// TIA Portal V17 export
// export: Created 2023-08-28T22:41:32.6164324Z, ExportSetting WithDefaults, DisplayName Totally Integrated Automation Portal, DisplayVersion V17 Update 5, DisplayName TIA Portal Openness, DisplayVersion V17 Update 5, DisplayName TIA Portal Teamcenter Gateway, DisplayVersion V17 Update 5, DisplayName TIA Portal Version Control Interface, DisplayVersion V17, DisplayName Simotion SCOUT TIA, DisplayVersion 5.4.3.0, DisplayName TIA Portal Test Suite Advanced, DisplayVersion V17 Update 1, DisplayName SIMOCODE ES, DisplayVersion V17 Update 5, DisplayName SINAMICS Startdrive Advanced, DisplayVersion V17 SP1, DisplayName SINAMICS Startdrive G130, G150, S120, S150, SINAMICS MV, S210, DisplayVersion V17 SP1, DisplayName SINAMICS Startdrive G110M, G120, G120C, G120D, G120P, G115D, DisplayVersion V17 SP1, DisplayName SIRIUS Safety ES, DisplayVersion V17 Update 5, DisplayName STEP 7 Professional, DisplayVersion V17 Update 5, DisplayName STEP 7 CFC, DisplayVersion V17 Update 1, DisplayName STEP 7 Safety, DisplayVersion V17, DisplayName WinCC Advanced, DisplayVersion V17 Update 5, DisplayName SIMATIC Visualization Architect, DisplayVersion V17 Update 5
DATA_BLOCK "n0005-zp001-el001-k40001_SN50_1"   // DB1001, F_DB
VERSION : 0.1
// stored: AutoNumber true, DBAccessibleFromOPCUA true, DBAccessibleFromWebserver true, InstanceOfName 00_Push-Button_Input, InstanceOfType FB
"00_Push-Button_Input"
   // VAR_INPUT
   //    IN_1 : Bool;
   //    IN_2 : Bool;
   //    IN_3 : Bool;
   //    IN_4 : Bool;
   //    ON_Tristate : Bool;
   //    ON_Lamp : Bool;
   //    Reset : Bool;
   //    REAC_DELAY { ExternalWritable := 'False'} : Time;
   //    Bypass_ET200 : Bool;
   // END_VAR
   // VAR_OUTPUT
   //    OUT_1 : Bool;
   //    OUT_2 : Bool;
   //    OUT_3 : Bool;
   //    OUT_4 : Bool;
   //    Diag_1 : Bool;
   //    Diag_2 : Bool;
   //    Diag_3 : Bool;
   //    Diag_4 : Bool;
   //    Lamp_1 : Bool;
   //    Lamp_2 : Bool;
   //    Lamp_3 : Bool;
   //    Lamp_4 : Bool;
   // END_VAR
   // VAR
   //    ESTOP_1 { S7_SetPoint := 'True'} : ESTOP1;
   //    ESTOP_2 { S7_SetPoint := 'True'} : ESTOP1;
   //    ESTOP_3 { S7_SetPoint := 'True'} : ESTOP1;
   //    ESTOP_4 { S7_SetPoint := 'True'} : ESTOP1;
   //    TON_1 { ExternalWritable := 'False'} : TON;
   //    TON_2 { ExternalWritable := 'False'} : TON;
   //    TON_3 { ExternalWritable := 'False'} : TON;
   //    TON_4 { ExternalWritable := 'False'} : TON;
   // END_VAR
BEGIN
END_DATA_BLOCK

DATA_BLOCK "n0013-uf317-xn10_SN50_1"   // DB1002, F_DB
VERSION : 0.1
// stored: AutoNumber true, DBAccessibleFromOPCUA true, DBAccessibleFromWebserver true, InstanceOfName 00_Push-Button_Input, InstanceOfType FB
"00_Push-Button_Input"
   // VAR_INPUT
   //    IN_1 : Bool;
   //    IN_2 : Bool;
   //    IN_3 : Bool;
   //    IN_4 : Bool;
   //    ON_Tristate : Bool;
   //    ON_Lamp : Bool;
   //    Reset : Bool;
   //    REAC_DELAY { ExternalWritable := 'False'} : Time;
   //    Bypass_ET200 : Bool;
   // END_VAR
   // VAR_OUTPUT
   //    OUT_1 : Bool;
   //    OUT_2 : Bool;
   //    OUT_3 : Bool;
   //    OUT_4 : Bool;
   //    Diag_1 : Bool;
   //    Diag_2 : Bool;
   //    Diag_3 : Bool;
   //    Diag_4 : Bool;
   //    Lamp_1 : Bool;
   //    Lamp_2 : Bool;
   //    Lamp_3 : Bool;
   //    Lamp_4 : Bool;
   // END_VAR
   // VAR
   //    ESTOP_1 { S7_SetPoint := 'True'} : ESTOP1;
   //    ESTOP_2 { S7_SetPoint := 'True'} : ESTOP1;
   //    ESTOP_3 { S7_SetPoint := 'True'} : ESTOP1;
   //    ESTOP_4 { S7_SetPoint := 'True'} : ESTOP1;
   //    TON_1 { ExternalWritable := 'False'} : TON;
   //    TON_2 { ExternalWritable := 'False'} : TON;
   //    TON_3 { ExternalWritable := 'False'} : TON;
   //    TON_4 { ExternalWritable := 'False'} : TON;
   // END_VAR
BEGIN
END_DATA_BLOCK

DATA_BLOCK "n0013-uf317-xn10_SN50_2"   // DB1003, F_DB
VERSION : 0.1
// stored: AutoNumber true, DBAccessibleFromOPCUA true, DBAccessibleFromWebserver true, InstanceOfName 00_Push-Button_Input, InstanceOfType FB
"00_Push-Button_Input"
   // VAR_INPUT
   //    IN_1 : Bool;
   //    IN_2 : Bool;
   //    IN_3 : Bool;
   //    IN_4 : Bool;
   //    ON_Tristate : Bool;
   //    ON_Lamp : Bool;
   //    Reset : Bool;
   //    REAC_DELAY { ExternalWritable := 'False'} : Time;
   //    Bypass_ET200 : Bool;
   // END_VAR
   // VAR_OUTPUT
   //    OUT_1 : Bool;
   //    OUT_2 : Bool;
   //    OUT_3 : Bool;
   //    OUT_4 : Bool;
   //    Diag_1 : Bool;
   //    Diag_2 : Bool;
   //    Diag_3 : Bool;
   //    Diag_4 : Bool;
   //    Lamp_1 : Bool;
   //    Lamp_2 : Bool;
   //    Lamp_3 : Bool;
   //    Lamp_4 : Bool;
   // END_VAR
   // VAR
   //    ESTOP_1 { S7_SetPoint := 'True'} : ESTOP1;
   //    ESTOP_2 { S7_SetPoint := 'True'} : ESTOP1;
   //    ESTOP_3 { S7_SetPoint := 'True'} : ESTOP1;
   //    ESTOP_4 { S7_SetPoint := 'True'} : ESTOP1;
   //    TON_1 { ExternalWritable := 'False'} : TON;
   //    TON_2 { ExternalWritable := 'False'} : TON;
   //    TON_3 { ExternalWritable := 'False'} : TON;
   //    TON_4 { ExternalWritable := 'False'} : TON;
   // END_VAR
BEGIN
END_DATA_BLOCK

DATA_BLOCK "n0015-uc16-el001-k30001_SN50_1"   // DB1004, F_DB
VERSION : 0.1
// stored: AutoNumber true, DBAccessibleFromOPCUA true, DBAccessibleFromWebserver true, InstanceOfName 00_Push-Button_Input, InstanceOfType FB
"00_Push-Button_Input"
   // VAR_INPUT
   //    IN_1 : Bool;
   //    IN_2 : Bool;
   //    IN_3 : Bool;
   //    IN_4 : Bool;
   //    ON_Tristate : Bool;
   //    ON_Lamp : Bool;
   //    Reset : Bool;
   //    REAC_DELAY { ExternalWritable := 'False'} : Time;
   //    Bypass_ET200 : Bool;
   // END_VAR
   // VAR_OUTPUT
   //    OUT_1 : Bool;
   //    OUT_2 : Bool;
   //    OUT_3 : Bool;
   //    OUT_4 : Bool;
   //    Diag_1 : Bool;
   //    Diag_2 : Bool;
   //    Diag_3 : Bool;
   //    Diag_4 : Bool;
   //    Lamp_1 : Bool;
   //    Lamp_2 : Bool;
   //    Lamp_3 : Bool;
   //    Lamp_4 : Bool;
   // END_VAR
   // VAR
   //    ESTOP_1 { S7_SetPoint := 'True'} : ESTOP1;
   //    ESTOP_2 { S7_SetPoint := 'True'} : ESTOP1;
   //    ESTOP_3 { S7_SetPoint := 'True'} : ESTOP1;
   //    ESTOP_4 { S7_SetPoint := 'True'} : ESTOP1;
   //    TON_1 { ExternalWritable := 'False'} : TON;
   //    TON_2 { ExternalWritable := 'False'} : TON;
   //    TON_3 { ExternalWritable := 'False'} : TON;
   //    TON_4 { ExternalWritable := 'False'} : TON;
   // END_VAR
BEGIN
END_DATA_BLOCK

DATA_BLOCK "n0015-uc16-el001-k30001_SN50_2"   // DB1005, F_DB
VERSION : 0.1
// stored: AutoNumber true, DBAccessibleFromOPCUA true, DBAccessibleFromWebserver true, InstanceOfName 00_Push-Button_Input, InstanceOfType FB
"00_Push-Button_Input"
   // VAR_INPUT
   //    IN_1 : Bool;
   //    IN_2 : Bool;
   //    IN_3 : Bool;
   //    IN_4 : Bool;
   //    ON_Tristate : Bool;
   //    ON_Lamp : Bool;
   //    Reset : Bool;
   //    REAC_DELAY { ExternalWritable := 'False'} : Time;
   //    Bypass_ET200 : Bool;
   // END_VAR
   // VAR_OUTPUT
   //    OUT_1 : Bool;
   //    OUT_2 : Bool;
   //    OUT_3 : Bool;
   //    OUT_4 : Bool;
   //    Diag_1 : Bool;
   //    Diag_2 : Bool;
   //    Diag_3 : Bool;
   //    Diag_4 : Bool;
   //    Lamp_1 : Bool;
   //    Lamp_2 : Bool;
   //    Lamp_3 : Bool;
   //    Lamp_4 : Bool;
   // END_VAR
   // VAR
   //    ESTOP_1 { S7_SetPoint := 'True'} : ESTOP1;
   //    ESTOP_2 { S7_SetPoint := 'True'} : ESTOP1;
   //    ESTOP_3 { S7_SetPoint := 'True'} : ESTOP1;
   //    ESTOP_4 { S7_SetPoint := 'True'} : ESTOP1;
   //    TON_1 { ExternalWritable := 'False'} : TON;
   //    TON_2 { ExternalWritable := 'False'} : TON;
   //    TON_3 { ExternalWritable := 'False'} : TON;
   //    TON_4 { ExternalWritable := 'False'} : TON;
   // END_VAR
BEGIN
END_DATA_BLOCK

DATA_BLOCK "n0015-uc16-el001-k30001_SN50_3"   // DB1006, F_DB
VERSION : 0.1
// stored: AutoNumber true, DBAccessibleFromOPCUA true, DBAccessibleFromWebserver true, InstanceOfName 00_Push-Button_Input, InstanceOfType FB
"00_Push-Button_Input"
   // VAR_INPUT
   //    IN_1 : Bool;
   //    IN_2 : Bool;
   //    IN_3 : Bool;
   //    IN_4 : Bool;
   //    ON_Tristate : Bool;
   //    ON_Lamp : Bool;
   //    Reset : Bool;
   //    REAC_DELAY { ExternalWritable := 'False'} : Time;
   //    Bypass_ET200 : Bool;
   // END_VAR
   // VAR_OUTPUT
   //    OUT_1 : Bool;
   //    OUT_2 : Bool;
   //    OUT_3 : Bool;
   //    OUT_4 : Bool;
   //    Diag_1 : Bool;
   //    Diag_2 : Bool;
   //    Diag_3 : Bool;
   //    Diag_4 : Bool;
   //    Lamp_1 : Bool;
   //    Lamp_2 : Bool;
   //    Lamp_3 : Bool;
   //    Lamp_4 : Bool;
   // END_VAR
   // VAR
   //    ESTOP_1 { S7_SetPoint := 'True'} : ESTOP1;
   //    ESTOP_2 { S7_SetPoint := 'True'} : ESTOP1;
   //    ESTOP_3 { S7_SetPoint := 'True'} : ESTOP1;
   //    ESTOP_4 { S7_SetPoint := 'True'} : ESTOP1;
   //    TON_1 { ExternalWritable := 'False'} : TON;
   //    TON_2 { ExternalWritable := 'False'} : TON;
   //    TON_3 { ExternalWritable := 'False'} : TON;
   //    TON_4 { ExternalWritable := 'False'} : TON;
   // END_VAR
BEGIN
END_DATA_BLOCK

DATA_BLOCK "n0016-uc164-xn10_SN50_1"   // DB1007, F_DB
VERSION : 0.1
// stored: AutoNumber true, DBAccessibleFromOPCUA true, DBAccessibleFromWebserver true, InstanceOfName 00_Push-Button_Input, InstanceOfType FB
"00_Push-Button_Input"
   // VAR_INPUT
   //    IN_1 : Bool;
   //    IN_2 : Bool;
   //    IN_3 : Bool;
   //    IN_4 : Bool;
   //    ON_Tristate : Bool;
   //    ON_Lamp : Bool;
   //    Reset : Bool;
   //    REAC_DELAY { ExternalWritable := 'False'} : Time;
   //    Bypass_ET200 : Bool;
   // END_VAR
   // VAR_OUTPUT
   //    OUT_1 : Bool;
   //    OUT_2 : Bool;
   //    OUT_3 : Bool;
   //    OUT_4 : Bool;
   //    Diag_1 : Bool;
   //    Diag_2 : Bool;
   //    Diag_3 : Bool;
   //    Diag_4 : Bool;
   //    Lamp_1 : Bool;
   //    Lamp_2 : Bool;
   //    Lamp_3 : Bool;
   //    Lamp_4 : Bool;
   // END_VAR
   // VAR
   //    ESTOP_1 { S7_SetPoint := 'True'} : ESTOP1;
   //    ESTOP_2 { S7_SetPoint := 'True'} : ESTOP1;
   //    ESTOP_3 { S7_SetPoint := 'True'} : ESTOP1;
   //    ESTOP_4 { S7_SetPoint := 'True'} : ESTOP1;
   //    TON_1 { ExternalWritable := 'False'} : TON;
   //    TON_2 { ExternalWritable := 'False'} : TON;
   //    TON_3 { ExternalWritable := 'False'} : TON;
   //    TON_4 { ExternalWritable := 'False'} : TON;
   // END_VAR
BEGIN
END_DATA_BLOCK

DATA_BLOCK "n0016-uc164-xn10_SN50_2"   // DB1008, F_DB
VERSION : 0.1
// stored: AutoNumber true, DBAccessibleFromOPCUA true, DBAccessibleFromWebserver true, InstanceOfName 00_Push-Button_Input, InstanceOfType FB
"00_Push-Button_Input"
   // VAR_INPUT
   //    IN_1 : Bool;
   //    IN_2 : Bool;
   //    IN_3 : Bool;
   //    IN_4 : Bool;
   //    ON_Tristate : Bool;
   //    ON_Lamp : Bool;
   //    Reset : Bool;
   //    REAC_DELAY { ExternalWritable := 'False'} : Time;
   //    Bypass_ET200 : Bool;
   // END_VAR
   // VAR_OUTPUT
   //    OUT_1 : Bool;
   //    OUT_2 : Bool;
   //    OUT_3 : Bool;
   //    OUT_4 : Bool;
   //    Diag_1 : Bool;
   //    Diag_2 : Bool;
   //    Diag_3 : Bool;
   //    Diag_4 : Bool;
   //    Lamp_1 : Bool;
   //    Lamp_2 : Bool;
   //    Lamp_3 : Bool;
   //    Lamp_4 : Bool;
   // END_VAR
   // VAR
   //    ESTOP_1 { S7_SetPoint := 'True'} : ESTOP1;
   //    ESTOP_2 { S7_SetPoint := 'True'} : ESTOP1;
   //    ESTOP_3 { S7_SetPoint := 'True'} : ESTOP1;
   //    ESTOP_4 { S7_SetPoint := 'True'} : ESTOP1;
   //    TON_1 { ExternalWritable := 'False'} : TON;
   //    TON_2 { ExternalWritable := 'False'} : TON;
   //    TON_3 { ExternalWritable := 'False'} : TON;
   //    TON_4 { ExternalWritable := 'False'} : TON;
   // END_VAR
BEGIN
END_DATA_BLOCK

DATA_BLOCK "n0020-uc15-el001-k30001_SN50_1"   // DB1009, F_DB
VERSION : 0.1
// stored: AutoNumber true, DBAccessibleFromOPCUA true, DBAccessibleFromWebserver true, InstanceOfName 00_Push-Button_Input, InstanceOfType FB
"00_Push-Button_Input"
   // VAR_INPUT
   //    IN_1 : Bool;
   //    IN_2 : Bool;
   //    IN_3 : Bool;
   //    IN_4 : Bool;
   //    ON_Tristate : Bool;
   //    ON_Lamp : Bool;
   //    Reset : Bool;
   //    REAC_DELAY { ExternalWritable := 'False'} : Time;
   //    Bypass_ET200 : Bool;
   // END_VAR
   // VAR_OUTPUT
   //    OUT_1 : Bool;
   //    OUT_2 : Bool;
   //    OUT_3 : Bool;
   //    OUT_4 : Bool;
   //    Diag_1 : Bool;
   //    Diag_2 : Bool;
   //    Diag_3 : Bool;
   //    Diag_4 : Bool;
   //    Lamp_1 : Bool;
   //    Lamp_2 : Bool;
   //    Lamp_3 : Bool;
   //    Lamp_4 : Bool;
   // END_VAR
   // VAR
   //    ESTOP_1 { S7_SetPoint := 'True'} : ESTOP1;
   //    ESTOP_2 { S7_SetPoint := 'True'} : ESTOP1;
   //    ESTOP_3 { S7_SetPoint := 'True'} : ESTOP1;
   //    ESTOP_4 { S7_SetPoint := 'True'} : ESTOP1;
   //    TON_1 { ExternalWritable := 'False'} : TON;
   //    TON_2 { ExternalWritable := 'False'} : TON;
   //    TON_3 { ExternalWritable := 'False'} : TON;
   //    TON_4 { ExternalWritable := 'False'} : TON;
   // END_VAR
BEGIN
END_DATA_BLOCK

DATA_BLOCK "n0020-uc15-el001-k30001_SN50_2"   // DB1010, F_DB
VERSION : 0.1
// stored: AutoNumber true, DBAccessibleFromOPCUA true, DBAccessibleFromWebserver true, InstanceOfName 00_Push-Button_Input, InstanceOfType FB
"00_Push-Button_Input"
   // VAR_INPUT
   //    IN_1 : Bool;
   //    IN_2 : Bool;
   //    IN_3 : Bool;
   //    IN_4 : Bool;
   //    ON_Tristate : Bool;
   //    ON_Lamp : Bool;
   //    Reset : Bool;
   //    REAC_DELAY { ExternalWritable := 'False'} : Time;
   //    Bypass_ET200 : Bool;
   // END_VAR
   // VAR_OUTPUT
   //    OUT_1 : Bool;
   //    OUT_2 : Bool;
   //    OUT_3 : Bool;
   //    OUT_4 : Bool;
   //    Diag_1 : Bool;
   //    Diag_2 : Bool;
   //    Diag_3 : Bool;
   //    Diag_4 : Bool;
   //    Lamp_1 : Bool;
   //    Lamp_2 : Bool;
   //    Lamp_3 : Bool;
   //    Lamp_4 : Bool;
   // END_VAR
   // VAR
   //    ESTOP_1 { S7_SetPoint := 'True'} : ESTOP1;
   //    ESTOP_2 { S7_SetPoint := 'True'} : ESTOP1;
   //    ESTOP_3 { S7_SetPoint := 'True'} : ESTOP1;
   //    ESTOP_4 { S7_SetPoint := 'True'} : ESTOP1;
   //    TON_1 { ExternalWritable := 'False'} : TON;
   //    TON_2 { ExternalWritable := 'False'} : TON;
   //    TON_3 { ExternalWritable := 'False'} : TON;
   //    TON_4 { ExternalWritable := 'False'} : TON;
   // END_VAR
BEGIN
END_DATA_BLOCK

DATA_BLOCK "n0020-uc15-el001-k30001_SN50_3"   // DB1011, F_DB
VERSION : 0.1
// stored: AutoNumber true, DBAccessibleFromOPCUA true, DBAccessibleFromWebserver true, InstanceOfName 00_Push-Button_Input, InstanceOfType FB
"00_Push-Button_Input"
   // VAR_INPUT
   //    IN_1 : Bool;
   //    IN_2 : Bool;
   //    IN_3 : Bool;
   //    IN_4 : Bool;
   //    ON_Tristate : Bool;
   //    ON_Lamp : Bool;
   //    Reset : Bool;
   //    REAC_DELAY { ExternalWritable := 'False'} : Time;
   //    Bypass_ET200 : Bool;
   // END_VAR
   // VAR_OUTPUT
   //    OUT_1 : Bool;
   //    OUT_2 : Bool;
   //    OUT_3 : Bool;
   //    OUT_4 : Bool;
   //    Diag_1 : Bool;
   //    Diag_2 : Bool;
   //    Diag_3 : Bool;
   //    Diag_4 : Bool;
   //    Lamp_1 : Bool;
   //    Lamp_2 : Bool;
   //    Lamp_3 : Bool;
   //    Lamp_4 : Bool;
   // END_VAR
   // VAR
   //    ESTOP_1 { S7_SetPoint := 'True'} : ESTOP1;
   //    ESTOP_2 { S7_SetPoint := 'True'} : ESTOP1;
   //    ESTOP_3 { S7_SetPoint := 'True'} : ESTOP1;
   //    ESTOP_4 { S7_SetPoint := 'True'} : ESTOP1;
   //    TON_1 { ExternalWritable := 'False'} : TON;
   //    TON_2 { ExternalWritable := 'False'} : TON;
   //    TON_3 { ExternalWritable := 'False'} : TON;
   //    TON_4 { ExternalWritable := 'False'} : TON;
   // END_VAR
BEGIN
END_DATA_BLOCK

DATA_BLOCK "n0023-uc154-xn10_SN50_1"   // DB1012, F_DB
VERSION : 0.1
// stored: AutoNumber true, DBAccessibleFromOPCUA true, DBAccessibleFromWebserver true, InstanceOfName 00_Push-Button_Input, InstanceOfType FB
"00_Push-Button_Input"
   // VAR_INPUT
   //    IN_1 : Bool;
   //    IN_2 : Bool;
   //    IN_3 : Bool;
   //    IN_4 : Bool;
   //    ON_Tristate : Bool;
   //    ON_Lamp : Bool;
   //    Reset : Bool;
   //    REAC_DELAY { ExternalWritable := 'False'} : Time;
   //    Bypass_ET200 : Bool;
   // END_VAR
   // VAR_OUTPUT
   //    OUT_1 : Bool;
   //    OUT_2 : Bool;
   //    OUT_3 : Bool;
   //    OUT_4 : Bool;
   //    Diag_1 : Bool;
   //    Diag_2 : Bool;
   //    Diag_3 : Bool;
   //    Diag_4 : Bool;
   //    Lamp_1 : Bool;
   //    Lamp_2 : Bool;
   //    Lamp_3 : Bool;
   //    Lamp_4 : Bool;
   // END_VAR
   // VAR
   //    ESTOP_1 { S7_SetPoint := 'True'} : ESTOP1;
   //    ESTOP_2 { S7_SetPoint := 'True'} : ESTOP1;
   //    ESTOP_3 { S7_SetPoint := 'True'} : ESTOP1;
   //    ESTOP_4 { S7_SetPoint := 'True'} : ESTOP1;
   //    TON_1 { ExternalWritable := 'False'} : TON;
   //    TON_2 { ExternalWritable := 'False'} : TON;
   //    TON_3 { ExternalWritable := 'False'} : TON;
   //    TON_4 { ExternalWritable := 'False'} : TON;
   // END_VAR
BEGIN
END_DATA_BLOCK

DATA_BLOCK "n0023-uc154-xn10_SN50_2"   // DB1013, F_DB
VERSION : 0.1
// stored: AutoNumber true, DBAccessibleFromOPCUA true, DBAccessibleFromWebserver true, InstanceOfName 00_Push-Button_Input, InstanceOfType FB
"00_Push-Button_Input"
   // VAR_INPUT
   //    IN_1 : Bool;
   //    IN_2 : Bool;
   //    IN_3 : Bool;
   //    IN_4 : Bool;
   //    ON_Tristate : Bool;
   //    ON_Lamp : Bool;
   //    Reset : Bool;
   //    REAC_DELAY { ExternalWritable := 'False'} : Time;
   //    Bypass_ET200 : Bool;
   // END_VAR
   // VAR_OUTPUT
   //    OUT_1 : Bool;
   //    OUT_2 : Bool;
   //    OUT_3 : Bool;
   //    OUT_4 : Bool;
   //    Diag_1 : Bool;
   //    Diag_2 : Bool;
   //    Diag_3 : Bool;
   //    Diag_4 : Bool;
   //    Lamp_1 : Bool;
   //    Lamp_2 : Bool;
   //    Lamp_3 : Bool;
   //    Lamp_4 : Bool;
   // END_VAR
   // VAR
   //    ESTOP_1 { S7_SetPoint := 'True'} : ESTOP1;
   //    ESTOP_2 { S7_SetPoint := 'True'} : ESTOP1;
   //    ESTOP_3 { S7_SetPoint := 'True'} : ESTOP1;
   //    ESTOP_4 { S7_SetPoint := 'True'} : ESTOP1;
   //    TON_1 { ExternalWritable := 'False'} : TON;
   //    TON_2 { ExternalWritable := 'False'} : TON;
   //    TON_3 { ExternalWritable := 'False'} : TON;
   //    TON_4 { ExternalWritable := 'False'} : TON;
   // END_VAR
BEGIN
END_DATA_BLOCK

DATA_BLOCK "n0021-icg11-el001-k30001_SN50_1"   // DB1014, F_DB
VERSION : 0.1
// stored: AutoNumber true, DBAccessibleFromOPCUA true, DBAccessibleFromWebserver true, InstanceOfName 00_Push-Button_Input, InstanceOfType FB
"00_Push-Button_Input"
   // VAR_INPUT
   //    IN_1 : Bool;
   //    IN_2 : Bool;
   //    IN_3 : Bool;
   //    IN_4 : Bool;
   //    ON_Tristate : Bool;
   //    ON_Lamp : Bool;
   //    Reset : Bool;
   //    REAC_DELAY { ExternalWritable := 'False'} : Time;
   //    Bypass_ET200 : Bool;
   // END_VAR
   // VAR_OUTPUT
   //    OUT_1 : Bool;
   //    OUT_2 : Bool;
   //    OUT_3 : Bool;
   //    OUT_4 : Bool;
   //    Diag_1 : Bool;
   //    Diag_2 : Bool;
   //    Diag_3 : Bool;
   //    Diag_4 : Bool;
   //    Lamp_1 : Bool;
   //    Lamp_2 : Bool;
   //    Lamp_3 : Bool;
   //    Lamp_4 : Bool;
   // END_VAR
   // VAR
   //    ESTOP_1 { S7_SetPoint := 'True'} : ESTOP1;
   //    ESTOP_2 { S7_SetPoint := 'True'} : ESTOP1;
   //    ESTOP_3 { S7_SetPoint := 'True'} : ESTOP1;
   //    ESTOP_4 { S7_SetPoint := 'True'} : ESTOP1;
   //    TON_1 { ExternalWritable := 'False'} : TON;
   //    TON_2 { ExternalWritable := 'False'} : TON;
   //    TON_3 { ExternalWritable := 'False'} : TON;
   //    TON_4 { ExternalWritable := 'False'} : TON;
   // END_VAR
BEGIN
END_DATA_BLOCK

DATA_BLOCK "n0021-icg11-el001-k30001_SN50_2"   // DB1015, F_DB
VERSION : 0.1
// stored: AutoNumber true, DBAccessibleFromOPCUA true, DBAccessibleFromWebserver true, InstanceOfName 00_Push-Button_Input, InstanceOfType FB
"00_Push-Button_Input"
   // VAR_INPUT
   //    IN_1 : Bool;
   //    IN_2 : Bool;
   //    IN_3 : Bool;
   //    IN_4 : Bool;
   //    ON_Tristate : Bool;
   //    ON_Lamp : Bool;
   //    Reset : Bool;
   //    REAC_DELAY { ExternalWritable := 'False'} : Time;
   //    Bypass_ET200 : Bool;
   // END_VAR
   // VAR_OUTPUT
   //    OUT_1 : Bool;
   //    OUT_2 : Bool;
   //    OUT_3 : Bool;
   //    OUT_4 : Bool;
   //    Diag_1 : Bool;
   //    Diag_2 : Bool;
   //    Diag_3 : Bool;
   //    Diag_4 : Bool;
   //    Lamp_1 : Bool;
   //    Lamp_2 : Bool;
   //    Lamp_3 : Bool;
   //    Lamp_4 : Bool;
   // END_VAR
   // VAR
   //    ESTOP_1 { S7_SetPoint := 'True'} : ESTOP1;
   //    ESTOP_2 { S7_SetPoint := 'True'} : ESTOP1;
   //    ESTOP_3 { S7_SetPoint := 'True'} : ESTOP1;
   //    ESTOP_4 { S7_SetPoint := 'True'} : ESTOP1;
   //    TON_1 { ExternalWritable := 'False'} : TON;
   //    TON_2 { ExternalWritable := 'False'} : TON;
   //    TON_3 { ExternalWritable := 'False'} : TON;
   //    TON_4 { ExternalWritable := 'False'} : TON;
   // END_VAR
BEGIN
END_DATA_BLOCK

DATA_BLOCK "n0021-icg11-el001-k30001_SN50_3"   // DB1016, F_DB
VERSION : 0.1
// stored: AutoNumber true, DBAccessibleFromOPCUA true, DBAccessibleFromWebserver true, InstanceOfName 00_Push-Button_Input, InstanceOfType FB
"00_Push-Button_Input"
   // VAR_INPUT
   //    IN_1 : Bool;
   //    IN_2 : Bool;
   //    IN_3 : Bool;
   //    IN_4 : Bool;
   //    ON_Tristate : Bool;
   //    ON_Lamp : Bool;
   //    Reset : Bool;
   //    REAC_DELAY { ExternalWritable := 'False'} : Time;
   //    Bypass_ET200 : Bool;
   // END_VAR
   // VAR_OUTPUT
   //    OUT_1 : Bool;
   //    OUT_2 : Bool;
   //    OUT_3 : Bool;
   //    OUT_4 : Bool;
   //    Diag_1 : Bool;
   //    Diag_2 : Bool;
   //    Diag_3 : Bool;
   //    Diag_4 : Bool;
   //    Lamp_1 : Bool;
   //    Lamp_2 : Bool;
   //    Lamp_3 : Bool;
   //    Lamp_4 : Bool;
   // END_VAR
   // VAR
   //    ESTOP_1 { S7_SetPoint := 'True'} : ESTOP1;
   //    ESTOP_2 { S7_SetPoint := 'True'} : ESTOP1;
   //    ESTOP_3 { S7_SetPoint := 'True'} : ESTOP1;
   //    ESTOP_4 { S7_SetPoint := 'True'} : ESTOP1;
   //    TON_1 { ExternalWritable := 'False'} : TON;
   //    TON_2 { ExternalWritable := 'False'} : TON;
   //    TON_3 { ExternalWritable := 'False'} : TON;
   //    TON_4 { ExternalWritable := 'False'} : TON;
   // END_VAR
BEGIN
END_DATA_BLOCK

DATA_BLOCK "n0021-icg11-el001-k30001_SN50_4"   // DB1017, F_DB
VERSION : 0.1
// stored: AutoNumber true, DBAccessibleFromOPCUA true, DBAccessibleFromWebserver true, InstanceOfName 00_Push-Button_Input, InstanceOfType FB
"00_Push-Button_Input"
   // VAR_INPUT
   //    IN_1 : Bool;
   //    IN_2 : Bool;
   //    IN_3 : Bool;
   //    IN_4 : Bool;
   //    ON_Tristate : Bool;
   //    ON_Lamp : Bool;
   //    Reset : Bool;
   //    REAC_DELAY { ExternalWritable := 'False'} : Time;
   //    Bypass_ET200 : Bool;
   // END_VAR
   // VAR_OUTPUT
   //    OUT_1 : Bool;
   //    OUT_2 : Bool;
   //    OUT_3 : Bool;
   //    OUT_4 : Bool;
   //    Diag_1 : Bool;
   //    Diag_2 : Bool;
   //    Diag_3 : Bool;
   //    Diag_4 : Bool;
   //    Lamp_1 : Bool;
   //    Lamp_2 : Bool;
   //    Lamp_3 : Bool;
   //    Lamp_4 : Bool;
   // END_VAR
   // VAR
   //    ESTOP_1 { S7_SetPoint := 'True'} : ESTOP1;
   //    ESTOP_2 { S7_SetPoint := 'True'} : ESTOP1;
   //    ESTOP_3 { S7_SetPoint := 'True'} : ESTOP1;
   //    ESTOP_4 { S7_SetPoint := 'True'} : ESTOP1;
   //    TON_1 { ExternalWritable := 'False'} : TON;
   //    TON_2 { ExternalWritable := 'False'} : TON;
   //    TON_3 { ExternalWritable := 'False'} : TON;
   //    TON_4 { ExternalWritable := 'False'} : TON;
   // END_VAR
BEGIN
END_DATA_BLOCK

DATA_BLOCK "n0022-icg21-el001-k30001_SN50_1"   // DB1018, F_DB
VERSION : 0.1
// stored: AutoNumber true, DBAccessibleFromOPCUA true, DBAccessibleFromWebserver true, InstanceOfName 00_Push-Button_Input, InstanceOfType FB
"00_Push-Button_Input"
   // VAR_INPUT
   //    IN_1 : Bool;
   //    IN_2 : Bool;
   //    IN_3 : Bool;
   //    IN_4 : Bool;
   //    ON_Tristate : Bool;
   //    ON_Lamp : Bool;
   //    Reset : Bool;
   //    REAC_DELAY { ExternalWritable := 'False'} : Time;
   //    Bypass_ET200 : Bool;
   // END_VAR
   // VAR_OUTPUT
   //    OUT_1 : Bool;
   //    OUT_2 : Bool;
   //    OUT_3 : Bool;
   //    OUT_4 : Bool;
   //    Diag_1 : Bool;
   //    Diag_2 : Bool;
   //    Diag_3 : Bool;
   //    Diag_4 : Bool;
   //    Lamp_1 : Bool;
   //    Lamp_2 : Bool;
   //    Lamp_3 : Bool;
   //    Lamp_4 : Bool;
   // END_VAR
   // VAR
   //    ESTOP_1 { S7_SetPoint := 'True'} : ESTOP1;
   //    ESTOP_2 { S7_SetPoint := 'True'} : ESTOP1;
   //    ESTOP_3 { S7_SetPoint := 'True'} : ESTOP1;
   //    ESTOP_4 { S7_SetPoint := 'True'} : ESTOP1;
   //    TON_1 { ExternalWritable := 'False'} : TON;
   //    TON_2 { ExternalWritable := 'False'} : TON;
   //    TON_3 { ExternalWritable := 'False'} : TON;
   //    TON_4 { ExternalWritable := 'False'} : TON;
   // END_VAR
BEGIN
END_DATA_BLOCK

DATA_BLOCK "n0022-icg21-el001-k30001_SN50_2"   // DB1019, F_DB
VERSION : 0.1
// stored: AutoNumber true, DBAccessibleFromOPCUA true, DBAccessibleFromWebserver true, InstanceOfName 00_Push-Button_Input, InstanceOfType FB
"00_Push-Button_Input"
   // VAR_INPUT
   //    IN_1 : Bool;
   //    IN_2 : Bool;
   //    IN_3 : Bool;
   //    IN_4 : Bool;
   //    ON_Tristate : Bool;
   //    ON_Lamp : Bool;
   //    Reset : Bool;
   //    REAC_DELAY { ExternalWritable := 'False'} : Time;
   //    Bypass_ET200 : Bool;
   // END_VAR
   // VAR_OUTPUT
   //    OUT_1 : Bool;
   //    OUT_2 : Bool;
   //    OUT_3 : Bool;
   //    OUT_4 : Bool;
   //    Diag_1 : Bool;
   //    Diag_2 : Bool;
   //    Diag_3 : Bool;
   //    Diag_4 : Bool;
   //    Lamp_1 : Bool;
   //    Lamp_2 : Bool;
   //    Lamp_3 : Bool;
   //    Lamp_4 : Bool;
   // END_VAR
   // VAR
   //    ESTOP_1 { S7_SetPoint := 'True'} : ESTOP1;
   //    ESTOP_2 { S7_SetPoint := 'True'} : ESTOP1;
   //    ESTOP_3 { S7_SetPoint := 'True'} : ESTOP1;
   //    ESTOP_4 { S7_SetPoint := 'True'} : ESTOP1;
   //    TON_1 { ExternalWritable := 'False'} : TON;
   //    TON_2 { ExternalWritable := 'False'} : TON;
   //    TON_3 { ExternalWritable := 'False'} : TON;
   //    TON_4 { ExternalWritable := 'False'} : TON;
   // END_VAR
BEGIN
END_DATA_BLOCK

DATA_BLOCK "n0025-uc14-el001-k30001_SN50_1"   // DB1020, F_DB
VERSION : 0.1
// stored: AutoNumber true, DBAccessibleFromOPCUA true, DBAccessibleFromWebserver true, InstanceOfName 00_Push-Button_Input, InstanceOfType FB
"00_Push-Button_Input"
   // VAR_INPUT
   //    IN_1 : Bool;
   //    IN_2 : Bool;
   //    IN_3 : Bool;
   //    IN_4 : Bool;
   //    ON_Tristate : Bool;
   //    ON_Lamp : Bool;
   //    Reset : Bool;
   //    REAC_DELAY { ExternalWritable := 'False'} : Time;
   //    Bypass_ET200 : Bool;
   // END_VAR
   // VAR_OUTPUT
   //    OUT_1 : Bool;
   //    OUT_2 : Bool;
   //    OUT_3 : Bool;
   //    OUT_4 : Bool;
   //    Diag_1 : Bool;
   //    Diag_2 : Bool;
   //    Diag_3 : Bool;
   //    Diag_4 : Bool;
   //    Lamp_1 : Bool;
   //    Lamp_2 : Bool;
   //    Lamp_3 : Bool;
   //    Lamp_4 : Bool;
   // END_VAR
   // VAR
   //    ESTOP_1 { S7_SetPoint := 'True'} : ESTOP1;
   //    ESTOP_2 { S7_SetPoint := 'True'} : ESTOP1;
   //    ESTOP_3 { S7_SetPoint := 'True'} : ESTOP1;
   //    ESTOP_4 { S7_SetPoint := 'True'} : ESTOP1;
   //    TON_1 { ExternalWritable := 'False'} : TON;
   //    TON_2 { ExternalWritable := 'False'} : TON;
   //    TON_3 { ExternalWritable := 'False'} : TON;
   //    TON_4 { ExternalWritable := 'False'} : TON;
   // END_VAR
BEGIN
END_DATA_BLOCK

DATA_BLOCK "n0025-uc14-el001-k30001_SN50_2"   // DB1021, F_DB
VERSION : 0.1
// stored: AutoNumber true, DBAccessibleFromOPCUA true, DBAccessibleFromWebserver true, InstanceOfName 00_Push-Button_Input, InstanceOfType FB
"00_Push-Button_Input"
   // VAR_INPUT
   //    IN_1 : Bool;
   //    IN_2 : Bool;
   //    IN_3 : Bool;
   //    IN_4 : Bool;
   //    ON_Tristate : Bool;
   //    ON_Lamp : Bool;
   //    Reset : Bool;
   //    REAC_DELAY { ExternalWritable := 'False'} : Time;
   //    Bypass_ET200 : Bool;
   // END_VAR
   // VAR_OUTPUT
   //    OUT_1 : Bool;
   //    OUT_2 : Bool;
   //    OUT_3 : Bool;
   //    OUT_4 : Bool;
   //    Diag_1 : Bool;
   //    Diag_2 : Bool;
   //    Diag_3 : Bool;
   //    Diag_4 : Bool;
   //    Lamp_1 : Bool;
   //    Lamp_2 : Bool;
   //    Lamp_3 : Bool;
   //    Lamp_4 : Bool;
   // END_VAR
   // VAR
   //    ESTOP_1 { S7_SetPoint := 'True'} : ESTOP1;
   //    ESTOP_2 { S7_SetPoint := 'True'} : ESTOP1;
   //    ESTOP_3 { S7_SetPoint := 'True'} : ESTOP1;
   //    ESTOP_4 { S7_SetPoint := 'True'} : ESTOP1;
   //    TON_1 { ExternalWritable := 'False'} : TON;
   //    TON_2 { ExternalWritable := 'False'} : TON;
   //    TON_3 { ExternalWritable := 'False'} : TON;
   //    TON_4 { ExternalWritable := 'False'} : TON;
   // END_VAR
BEGIN
END_DATA_BLOCK

DATA_BLOCK "n0025-uc14-el001-k30001_SN50_3"   // DB1022, F_DB
VERSION : 0.1
// stored: AutoNumber true, DBAccessibleFromOPCUA true, DBAccessibleFromWebserver true, InstanceOfName 00_Push-Button_Input, InstanceOfType FB
"00_Push-Button_Input"
   // VAR_INPUT
   //    IN_1 : Bool;
   //    IN_2 : Bool;
   //    IN_3 : Bool;
   //    IN_4 : Bool;
   //    ON_Tristate : Bool;
   //    ON_Lamp : Bool;
   //    Reset : Bool;
   //    REAC_DELAY { ExternalWritable := 'False'} : Time;
   //    Bypass_ET200 : Bool;
   // END_VAR
   // VAR_OUTPUT
   //    OUT_1 : Bool;
   //    OUT_2 : Bool;
   //    OUT_3 : Bool;
   //    OUT_4 : Bool;
   //    Diag_1 : Bool;
   //    Diag_2 : Bool;
   //    Diag_3 : Bool;
   //    Diag_4 : Bool;
   //    Lamp_1 : Bool;
   //    Lamp_2 : Bool;
   //    Lamp_3 : Bool;
   //    Lamp_4 : Bool;
   // END_VAR
   // VAR
   //    ESTOP_1 { S7_SetPoint := 'True'} : ESTOP1;
   //    ESTOP_2 { S7_SetPoint := 'True'} : ESTOP1;
   //    ESTOP_3 { S7_SetPoint := 'True'} : ESTOP1;
   //    ESTOP_4 { S7_SetPoint := 'True'} : ESTOP1;
   //    TON_1 { ExternalWritable := 'False'} : TON;
   //    TON_2 { ExternalWritable := 'False'} : TON;
   //    TON_3 { ExternalWritable := 'False'} : TON;
   //    TON_4 { ExternalWritable := 'False'} : TON;
   // END_VAR
BEGIN
END_DATA_BLOCK

DATA_BLOCK "n0026-uc144-xn10_SN50_1"   // DB1023, F_DB
VERSION : 0.1
// stored: AutoNumber true, DBAccessibleFromOPCUA true, DBAccessibleFromWebserver true, InstanceOfName 00_Push-Button_Input, InstanceOfType FB
"00_Push-Button_Input"
   // VAR_INPUT
   //    IN_1 : Bool;
   //    IN_2 : Bool;
   //    IN_3 : Bool;
   //    IN_4 : Bool;
   //    ON_Tristate : Bool;
   //    ON_Lamp : Bool;
   //    Reset : Bool;
   //    REAC_DELAY { ExternalWritable := 'False'} : Time;
   //    Bypass_ET200 : Bool;
   // END_VAR
   // VAR_OUTPUT
   //    OUT_1 : Bool;
   //    OUT_2 : Bool;
   //    OUT_3 : Bool;
   //    OUT_4 : Bool;
   //    Diag_1 : Bool;
   //    Diag_2 : Bool;
   //    Diag_3 : Bool;
   //    Diag_4 : Bool;
   //    Lamp_1 : Bool;
   //    Lamp_2 : Bool;
   //    Lamp_3 : Bool;
   //    Lamp_4 : Bool;
   // END_VAR
   // VAR
   //    ESTOP_1 { S7_SetPoint := 'True'} : ESTOP1;
   //    ESTOP_2 { S7_SetPoint := 'True'} : ESTOP1;
   //    ESTOP_3 { S7_SetPoint := 'True'} : ESTOP1;
   //    ESTOP_4 { S7_SetPoint := 'True'} : ESTOP1;
   //    TON_1 { ExternalWritable := 'False'} : TON;
   //    TON_2 { ExternalWritable := 'False'} : TON;
   //    TON_3 { ExternalWritable := 'False'} : TON;
   //    TON_4 { ExternalWritable := 'False'} : TON;
   // END_VAR
BEGIN
END_DATA_BLOCK

DATA_BLOCK "n0026-uc144-xn10_SN50_2"   // DB1024, F_DB
VERSION : 0.1
// stored: AutoNumber true, DBAccessibleFromOPCUA true, DBAccessibleFromWebserver true, InstanceOfName 00_Push-Button_Input, InstanceOfType FB
"00_Push-Button_Input"
   // VAR_INPUT
   //    IN_1 : Bool;
   //    IN_2 : Bool;
   //    IN_3 : Bool;
   //    IN_4 : Bool;
   //    ON_Tristate : Bool;
   //    ON_Lamp : Bool;
   //    Reset : Bool;
   //    REAC_DELAY { ExternalWritable := 'False'} : Time;
   //    Bypass_ET200 : Bool;
   // END_VAR
   // VAR_OUTPUT
   //    OUT_1 : Bool;
   //    OUT_2 : Bool;
   //    OUT_3 : Bool;
   //    OUT_4 : Bool;
   //    Diag_1 : Bool;
   //    Diag_2 : Bool;
   //    Diag_3 : Bool;
   //    Diag_4 : Bool;
   //    Lamp_1 : Bool;
   //    Lamp_2 : Bool;
   //    Lamp_3 : Bool;
   //    Lamp_4 : Bool;
   // END_VAR
   // VAR
   //    ESTOP_1 { S7_SetPoint := 'True'} : ESTOP1;
   //    ESTOP_2 { S7_SetPoint := 'True'} : ESTOP1;
   //    ESTOP_3 { S7_SetPoint := 'True'} : ESTOP1;
   //    ESTOP_4 { S7_SetPoint := 'True'} : ESTOP1;
   //    TON_1 { ExternalWritable := 'False'} : TON;
   //    TON_2 { ExternalWritable := 'False'} : TON;
   //    TON_3 { ExternalWritable := 'False'} : TON;
   //    TON_4 { ExternalWritable := 'False'} : TON;
   // END_VAR
BEGIN
END_DATA_BLOCK

DATA_BLOCK "n0038-uc1-el001-k30001_SN50_1"   // DB1025, F_DB
VERSION : 0.1
// stored: AutoNumber true, DBAccessibleFromOPCUA true, DBAccessibleFromWebserver true, InstanceOfName 00_Push-Button_Input, InstanceOfType FB
"00_Push-Button_Input"
   // VAR_INPUT
   //    IN_1 : Bool;
   //    IN_2 : Bool;
   //    IN_3 : Bool;
   //    IN_4 : Bool;
   //    ON_Tristate : Bool;
   //    ON_Lamp : Bool;
   //    Reset : Bool;
   //    REAC_DELAY { ExternalWritable := 'False'} : Time;
   //    Bypass_ET200 : Bool;
   // END_VAR
   // VAR_OUTPUT
   //    OUT_1 : Bool;
   //    OUT_2 : Bool;
   //    OUT_3 : Bool;
   //    OUT_4 : Bool;
   //    Diag_1 : Bool;
   //    Diag_2 : Bool;
   //    Diag_3 : Bool;
   //    Diag_4 : Bool;
   //    Lamp_1 : Bool;
   //    Lamp_2 : Bool;
   //    Lamp_3 : Bool;
   //    Lamp_4 : Bool;
   // END_VAR
   // VAR
   //    ESTOP_1 { S7_SetPoint := 'True'} : ESTOP1;
   //    ESTOP_2 { S7_SetPoint := 'True'} : ESTOP1;
   //    ESTOP_3 { S7_SetPoint := 'True'} : ESTOP1;
   //    ESTOP_4 { S7_SetPoint := 'True'} : ESTOP1;
   //    TON_1 { ExternalWritable := 'False'} : TON;
   //    TON_2 { ExternalWritable := 'False'} : TON;
   //    TON_3 { ExternalWritable := 'False'} : TON;
   //    TON_4 { ExternalWritable := 'False'} : TON;
   // END_VAR
BEGIN
END_DATA_BLOCK

DATA_BLOCK "n0041-uf31-el002-k30001_SN50_1"   // DB1026, F_DB
VERSION : 0.1
// stored: AutoNumber true, DBAccessibleFromOPCUA true, DBAccessibleFromWebserver true, InstanceOfName 00_Push-Button_Input, InstanceOfType FB
"00_Push-Button_Input"
   // VAR_INPUT
   //    IN_1 : Bool;
   //    IN_2 : Bool;
   //    IN_3 : Bool;
   //    IN_4 : Bool;
   //    ON_Tristate : Bool;
   //    ON_Lamp : Bool;
   //    Reset : Bool;
   //    REAC_DELAY { ExternalWritable := 'False'} : Time;
   //    Bypass_ET200 : Bool;
   // END_VAR
   // VAR_OUTPUT
   //    OUT_1 : Bool;
   //    OUT_2 : Bool;
   //    OUT_3 : Bool;
   //    OUT_4 : Bool;
   //    Diag_1 : Bool;
   //    Diag_2 : Bool;
   //    Diag_3 : Bool;
   //    Diag_4 : Bool;
   //    Lamp_1 : Bool;
   //    Lamp_2 : Bool;
   //    Lamp_3 : Bool;
   //    Lamp_4 : Bool;
   // END_VAR
   // VAR
   //    ESTOP_1 { S7_SetPoint := 'True'} : ESTOP1;
   //    ESTOP_2 { S7_SetPoint := 'True'} : ESTOP1;
   //    ESTOP_3 { S7_SetPoint := 'True'} : ESTOP1;
   //    ESTOP_4 { S7_SetPoint := 'True'} : ESTOP1;
   //    TON_1 { ExternalWritable := 'False'} : TON;
   //    TON_2 { ExternalWritable := 'False'} : TON;
   //    TON_3 { ExternalWritable := 'False'} : TON;
   //    TON_4 { ExternalWritable := 'False'} : TON;
   // END_VAR
BEGIN
END_DATA_BLOCK

DATA_BLOCK "n0044-ct1-el001-k30001_SN50_1"   // DB1027, F_DB
VERSION : 0.1
// stored: AutoNumber true, DBAccessibleFromOPCUA true, DBAccessibleFromWebserver true, InstanceOfName 00_Push-Button_Input, InstanceOfType FB
"00_Push-Button_Input"
   // VAR_INPUT
   //    IN_1 : Bool;
   //    IN_2 : Bool;
   //    IN_3 : Bool;
   //    IN_4 : Bool;
   //    ON_Tristate : Bool;
   //    ON_Lamp : Bool;
   //    Reset : Bool;
   //    REAC_DELAY { ExternalWritable := 'False'} : Time;
   //    Bypass_ET200 : Bool;
   // END_VAR
   // VAR_OUTPUT
   //    OUT_1 : Bool;
   //    OUT_2 : Bool;
   //    OUT_3 : Bool;
   //    OUT_4 : Bool;
   //    Diag_1 : Bool;
   //    Diag_2 : Bool;
   //    Diag_3 : Bool;
   //    Diag_4 : Bool;
   //    Lamp_1 : Bool;
   //    Lamp_2 : Bool;
   //    Lamp_3 : Bool;
   //    Lamp_4 : Bool;
   // END_VAR
   // VAR
   //    ESTOP_1 { S7_SetPoint := 'True'} : ESTOP1;
   //    ESTOP_2 { S7_SetPoint := 'True'} : ESTOP1;
   //    ESTOP_3 { S7_SetPoint := 'True'} : ESTOP1;
   //    ESTOP_4 { S7_SetPoint := 'True'} : ESTOP1;
   //    TON_1 { ExternalWritable := 'False'} : TON;
   //    TON_2 { ExternalWritable := 'False'} : TON;
   //    TON_3 { ExternalWritable := 'False'} : TON;
   //    TON_4 { ExternalWritable := 'False'} : TON;
   // END_VAR
BEGIN
END_DATA_BLOCK

DATA_BLOCK "n0044-ct1-el001-k30001_SN50_2"   // DB1028, F_DB
VERSION : 0.1
// stored: AutoNumber true, DBAccessibleFromOPCUA true, DBAccessibleFromWebserver true, InstanceOfName 00_Push-Button_Input, InstanceOfType FB
"00_Push-Button_Input"
   // VAR_INPUT
   //    IN_1 : Bool;
   //    IN_2 : Bool;
   //    IN_3 : Bool;
   //    IN_4 : Bool;
   //    ON_Tristate : Bool;
   //    ON_Lamp : Bool;
   //    Reset : Bool;
   //    REAC_DELAY { ExternalWritable := 'False'} : Time;
   //    Bypass_ET200 : Bool;
   // END_VAR
   // VAR_OUTPUT
   //    OUT_1 : Bool;
   //    OUT_2 : Bool;
   //    OUT_3 : Bool;
   //    OUT_4 : Bool;
   //    Diag_1 : Bool;
   //    Diag_2 : Bool;
   //    Diag_3 : Bool;
   //    Diag_4 : Bool;
   //    Lamp_1 : Bool;
   //    Lamp_2 : Bool;
   //    Lamp_3 : Bool;
   //    Lamp_4 : Bool;
   // END_VAR
   // VAR
   //    ESTOP_1 { S7_SetPoint := 'True'} : ESTOP1;
   //    ESTOP_2 { S7_SetPoint := 'True'} : ESTOP1;
   //    ESTOP_3 { S7_SetPoint := 'True'} : ESTOP1;
   //    ESTOP_4 { S7_SetPoint := 'True'} : ESTOP1;
   //    TON_1 { ExternalWritable := 'False'} : TON;
   //    TON_2 { ExternalWritable := 'False'} : TON;
   //    TON_3 { ExternalWritable := 'False'} : TON;
   //    TON_4 { ExternalWritable := 'False'} : TON;
   // END_VAR
BEGIN
END_DATA_BLOCK

DATA_BLOCK "n0044-ct1-el001-k30001_SN50_3"   // DB1029, F_DB
VERSION : 0.1
// stored: AutoNumber true, DBAccessibleFromOPCUA true, DBAccessibleFromWebserver true, InstanceOfName 00_Push-Button_Input, InstanceOfType FB
"00_Push-Button_Input"
   // VAR_INPUT
   //    IN_1 : Bool;
   //    IN_2 : Bool;
   //    IN_3 : Bool;
   //    IN_4 : Bool;
   //    ON_Tristate : Bool;
   //    ON_Lamp : Bool;
   //    Reset : Bool;
   //    REAC_DELAY { ExternalWritable := 'False'} : Time;
   //    Bypass_ET200 : Bool;
   // END_VAR
   // VAR_OUTPUT
   //    OUT_1 : Bool;
   //    OUT_2 : Bool;
   //    OUT_3 : Bool;
   //    OUT_4 : Bool;
   //    Diag_1 : Bool;
   //    Diag_2 : Bool;
   //    Diag_3 : Bool;
   //    Diag_4 : Bool;
   //    Lamp_1 : Bool;
   //    Lamp_2 : Bool;
   //    Lamp_3 : Bool;
   //    Lamp_4 : Bool;
   // END_VAR
   // VAR
   //    ESTOP_1 { S7_SetPoint := 'True'} : ESTOP1;
   //    ESTOP_2 { S7_SetPoint := 'True'} : ESTOP1;
   //    ESTOP_3 { S7_SetPoint := 'True'} : ESTOP1;
   //    ESTOP_4 { S7_SetPoint := 'True'} : ESTOP1;
   //    TON_1 { ExternalWritable := 'False'} : TON;
   //    TON_2 { ExternalWritable := 'False'} : TON;
   //    TON_3 { ExternalWritable := 'False'} : TON;
   //    TON_4 { ExternalWritable := 'False'} : TON;
   // END_VAR
BEGIN
END_DATA_BLOCK

DATA_BLOCK "n0044-ct1-el001-k30001_SN50_4"   // DB1030, F_DB
VERSION : 0.1
// stored: AutoNumber true, DBAccessibleFromOPCUA true, DBAccessibleFromWebserver true, InstanceOfName 00_Push-Button_Input, InstanceOfType FB
"00_Push-Button_Input"
   // VAR_INPUT
   //    IN_1 : Bool;
   //    IN_2 : Bool;
   //    IN_3 : Bool;
   //    IN_4 : Bool;
   //    ON_Tristate : Bool;
   //    ON_Lamp : Bool;
   //    Reset : Bool;
   //    REAC_DELAY { ExternalWritable := 'False'} : Time;
   //    Bypass_ET200 : Bool;
   // END_VAR
   // VAR_OUTPUT
   //    OUT_1 : Bool;
   //    OUT_2 : Bool;
   //    OUT_3 : Bool;
   //    OUT_4 : Bool;
   //    Diag_1 : Bool;
   //    Diag_2 : Bool;
   //    Diag_3 : Bool;
   //    Diag_4 : Bool;
   //    Lamp_1 : Bool;
   //    Lamp_2 : Bool;
   //    Lamp_3 : Bool;
   //    Lamp_4 : Bool;
   // END_VAR
   // VAR
   //    ESTOP_1 { S7_SetPoint := 'True'} : ESTOP1;
   //    ESTOP_2 { S7_SetPoint := 'True'} : ESTOP1;
   //    ESTOP_3 { S7_SetPoint := 'True'} : ESTOP1;
   //    ESTOP_4 { S7_SetPoint := 'True'} : ESTOP1;
   //    TON_1 { ExternalWritable := 'False'} : TON;
   //    TON_2 { ExternalWritable := 'False'} : TON;
   //    TON_3 { ExternalWritable := 'False'} : TON;
   //    TON_4 { ExternalWritable := 'False'} : TON;
   // END_VAR
BEGIN
END_DATA_BLOCK

DATA_BLOCK "n0045-ct1-el002-k30001_SN50_1"   // DB1031, F_DB
VERSION : 0.1
// stored: AutoNumber true, DBAccessibleFromOPCUA true, DBAccessibleFromWebserver true, InstanceOfName 00_Push-Button_Input, InstanceOfType FB
"00_Push-Button_Input"
   // VAR_INPUT
   //    IN_1 : Bool;
   //    IN_2 : Bool;
   //    IN_3 : Bool;
   //    IN_4 : Bool;
   //    ON_Tristate : Bool;
   //    ON_Lamp : Bool;
   //    Reset : Bool;
   //    REAC_DELAY { ExternalWritable := 'False'} : Time;
   //    Bypass_ET200 : Bool;
   // END_VAR
   // VAR_OUTPUT
   //    OUT_1 : Bool;
   //    OUT_2 : Bool;
   //    OUT_3 : Bool;
   //    OUT_4 : Bool;
   //    Diag_1 : Bool;
   //    Diag_2 : Bool;
   //    Diag_3 : Bool;
   //    Diag_4 : Bool;
   //    Lamp_1 : Bool;
   //    Lamp_2 : Bool;
   //    Lamp_3 : Bool;
   //    Lamp_4 : Bool;
   // END_VAR
   // VAR
   //    ESTOP_1 { S7_SetPoint := 'True'} : ESTOP1;
   //    ESTOP_2 { S7_SetPoint := 'True'} : ESTOP1;
   //    ESTOP_3 { S7_SetPoint := 'True'} : ESTOP1;
   //    ESTOP_4 { S7_SetPoint := 'True'} : ESTOP1;
   //    TON_1 { ExternalWritable := 'False'} : TON;
   //    TON_2 { ExternalWritable := 'False'} : TON;
   //    TON_3 { ExternalWritable := 'False'} : TON;
   //    TON_4 { ExternalWritable := 'False'} : TON;
   // END_VAR
BEGIN
END_DATA_BLOCK

DATA_BLOCK "n0045-ct1-el002-k30001_SN50_2"   // DB1032, F_DB
VERSION : 0.1
// stored: AutoNumber true, DBAccessibleFromOPCUA true, DBAccessibleFromWebserver true, InstanceOfName 00_Push-Button_Input, InstanceOfType FB
"00_Push-Button_Input"
   // VAR_INPUT
   //    IN_1 : Bool;
   //    IN_2 : Bool;
   //    IN_3 : Bool;
   //    IN_4 : Bool;
   //    ON_Tristate : Bool;
   //    ON_Lamp : Bool;
   //    Reset : Bool;
   //    REAC_DELAY { ExternalWritable := 'False'} : Time;
   //    Bypass_ET200 : Bool;
   // END_VAR
   // VAR_OUTPUT
   //    OUT_1 : Bool;
   //    OUT_2 : Bool;
   //    OUT_3 : Bool;
   //    OUT_4 : Bool;
   //    Diag_1 : Bool;
   //    Diag_2 : Bool;
   //    Diag_3 : Bool;
   //    Diag_4 : Bool;
   //    Lamp_1 : Bool;
   //    Lamp_2 : Bool;
   //    Lamp_3 : Bool;
   //    Lamp_4 : Bool;
   // END_VAR
   // VAR
   //    ESTOP_1 { S7_SetPoint := 'True'} : ESTOP1;
   //    ESTOP_2 { S7_SetPoint := 'True'} : ESTOP1;
   //    ESTOP_3 { S7_SetPoint := 'True'} : ESTOP1;
   //    ESTOP_4 { S7_SetPoint := 'True'} : ESTOP1;
   //    TON_1 { ExternalWritable := 'False'} : TON;
   //    TON_2 { ExternalWritable := 'False'} : TON;
   //    TON_3 { ExternalWritable := 'False'} : TON;
   //    TON_4 { ExternalWritable := 'False'} : TON;
   // END_VAR
BEGIN
END_DATA_BLOCK

DATA_BLOCK "n0045-ct1-el002-k30001_SN50_3"   // DB1033, F_DB
VERSION : 0.1
// stored: AutoNumber true, DBAccessibleFromOPCUA true, DBAccessibleFromWebserver true, InstanceOfName 00_Push-Button_Input, InstanceOfType FB
"00_Push-Button_Input"
   // VAR_INPUT
   //    IN_1 : Bool;
   //    IN_2 : Bool;
   //    IN_3 : Bool;
   //    IN_4 : Bool;
   //    ON_Tristate : Bool;
   //    ON_Lamp : Bool;
   //    Reset : Bool;
   //    REAC_DELAY { ExternalWritable := 'False'} : Time;
   //    Bypass_ET200 : Bool;
   // END_VAR
   // VAR_OUTPUT
   //    OUT_1 : Bool;
   //    OUT_2 : Bool;
   //    OUT_3 : Bool;
   //    OUT_4 : Bool;
   //    Diag_1 : Bool;
   //    Diag_2 : Bool;
   //    Diag_3 : Bool;
   //    Diag_4 : Bool;
   //    Lamp_1 : Bool;
   //    Lamp_2 : Bool;
   //    Lamp_3 : Bool;
   //    Lamp_4 : Bool;
   // END_VAR
   // VAR
   //    ESTOP_1 { S7_SetPoint := 'True'} : ESTOP1;
   //    ESTOP_2 { S7_SetPoint := 'True'} : ESTOP1;
   //    ESTOP_3 { S7_SetPoint := 'True'} : ESTOP1;
   //    ESTOP_4 { S7_SetPoint := 'True'} : ESTOP1;
   //    TON_1 { ExternalWritable := 'False'} : TON;
   //    TON_2 { ExternalWritable := 'False'} : TON;
   //    TON_3 { ExternalWritable := 'False'} : TON;
   //    TON_4 { ExternalWritable := 'False'} : TON;
   // END_VAR
BEGIN
END_DATA_BLOCK

DATA_BLOCK "n0045-ct1-el002-k30001_SN50_4"   // DB1034, F_DB
VERSION : 0.1
// stored: AutoNumber true, DBAccessibleFromOPCUA true, DBAccessibleFromWebserver true, InstanceOfName 00_Push-Button_Input, InstanceOfType FB
"00_Push-Button_Input"
   // VAR_INPUT
   //    IN_1 : Bool;
   //    IN_2 : Bool;
   //    IN_3 : Bool;
   //    IN_4 : Bool;
   //    ON_Tristate : Bool;
   //    ON_Lamp : Bool;
   //    Reset : Bool;
   //    REAC_DELAY { ExternalWritable := 'False'} : Time;
   //    Bypass_ET200 : Bool;
   // END_VAR
   // VAR_OUTPUT
   //    OUT_1 : Bool;
   //    OUT_2 : Bool;
   //    OUT_3 : Bool;
   //    OUT_4 : Bool;
   //    Diag_1 : Bool;
   //    Diag_2 : Bool;
   //    Diag_3 : Bool;
   //    Diag_4 : Bool;
   //    Lamp_1 : Bool;
   //    Lamp_2 : Bool;
   //    Lamp_3 : Bool;
   //    Lamp_4 : Bool;
   // END_VAR
   // VAR
   //    ESTOP_1 { S7_SetPoint := 'True'} : ESTOP1;
   //    ESTOP_2 { S7_SetPoint := 'True'} : ESTOP1;
   //    ESTOP_3 { S7_SetPoint := 'True'} : ESTOP1;
   //    ESTOP_4 { S7_SetPoint := 'True'} : ESTOP1;
   //    TON_1 { ExternalWritable := 'False'} : TON;
   //    TON_2 { ExternalWritable := 'False'} : TON;
   //    TON_3 { ExternalWritable := 'False'} : TON;
   //    TON_4 { ExternalWritable := 'False'} : TON;
   // END_VAR
BEGIN
END_DATA_BLOCK

DATA_BLOCK "n0045-ct1-el002-k30001_SN50_5"   // DB1035, F_DB
VERSION : 0.1
// stored: AutoNumber true, DBAccessibleFromOPCUA true, DBAccessibleFromWebserver true, InstanceOfName 00_Push-Button_Input, InstanceOfType FB
"00_Push-Button_Input"
   // VAR_INPUT
   //    IN_1 : Bool;
   //    IN_2 : Bool;
   //    IN_3 : Bool;
   //    IN_4 : Bool;
   //    ON_Tristate : Bool;
   //    ON_Lamp : Bool;
   //    Reset : Bool;
   //    REAC_DELAY { ExternalWritable := 'False'} : Time;
   //    Bypass_ET200 : Bool;
   // END_VAR
   // VAR_OUTPUT
   //    OUT_1 : Bool;
   //    OUT_2 : Bool;
   //    OUT_3 : Bool;
   //    OUT_4 : Bool;
   //    Diag_1 : Bool;
   //    Diag_2 : Bool;
   //    Diag_3 : Bool;
   //    Diag_4 : Bool;
   //    Lamp_1 : Bool;
   //    Lamp_2 : Bool;
   //    Lamp_3 : Bool;
   //    Lamp_4 : Bool;
   // END_VAR
   // VAR
   //    ESTOP_1 { S7_SetPoint := 'True'} : ESTOP1;
   //    ESTOP_2 { S7_SetPoint := 'True'} : ESTOP1;
   //    ESTOP_3 { S7_SetPoint := 'True'} : ESTOP1;
   //    ESTOP_4 { S7_SetPoint := 'True'} : ESTOP1;
   //    TON_1 { ExternalWritable := 'False'} : TON;
   //    TON_2 { ExternalWritable := 'False'} : TON;
   //    TON_3 { ExternalWritable := 'False'} : TON;
   //    TON_4 { ExternalWritable := 'False'} : TON;
   // END_VAR
BEGIN
END_DATA_BLOCK

DATA_BLOCK "n0046-ct1-el003-k30001_SN50_1"   // DB1036, F_DB
VERSION : 0.1
// stored: AutoNumber true, DBAccessibleFromOPCUA true, DBAccessibleFromWebserver true, InstanceOfName 00_Push-Button_Input, InstanceOfType FB
"00_Push-Button_Input"
   // VAR_INPUT
   //    IN_1 : Bool;
   //    IN_2 : Bool;
   //    IN_3 : Bool;
   //    IN_4 : Bool;
   //    ON_Tristate : Bool;
   //    ON_Lamp : Bool;
   //    Reset : Bool;
   //    REAC_DELAY { ExternalWritable := 'False'} : Time;
   //    Bypass_ET200 : Bool;
   // END_VAR
   // VAR_OUTPUT
   //    OUT_1 : Bool;
   //    OUT_2 : Bool;
   //    OUT_3 : Bool;
   //    OUT_4 : Bool;
   //    Diag_1 : Bool;
   //    Diag_2 : Bool;
   //    Diag_3 : Bool;
   //    Diag_4 : Bool;
   //    Lamp_1 : Bool;
   //    Lamp_2 : Bool;
   //    Lamp_3 : Bool;
   //    Lamp_4 : Bool;
   // END_VAR
   // VAR
   //    ESTOP_1 { S7_SetPoint := 'True'} : ESTOP1;
   //    ESTOP_2 { S7_SetPoint := 'True'} : ESTOP1;
   //    ESTOP_3 { S7_SetPoint := 'True'} : ESTOP1;
   //    ESTOP_4 { S7_SetPoint := 'True'} : ESTOP1;
   //    TON_1 { ExternalWritable := 'False'} : TON;
   //    TON_2 { ExternalWritable := 'False'} : TON;
   //    TON_3 { ExternalWritable := 'False'} : TON;
   //    TON_4 { ExternalWritable := 'False'} : TON;
   // END_VAR
BEGIN
END_DATA_BLOCK

DATA_BLOCK "n0046-ct1-el003-k30001_SN50_2"   // DB1037, F_DB
VERSION : 0.1
// stored: AutoNumber true, DBAccessibleFromOPCUA true, DBAccessibleFromWebserver true, InstanceOfName 00_Push-Button_Input, InstanceOfType FB
"00_Push-Button_Input"
   // VAR_INPUT
   //    IN_1 : Bool;
   //    IN_2 : Bool;
   //    IN_3 : Bool;
   //    IN_4 : Bool;
   //    ON_Tristate : Bool;
   //    ON_Lamp : Bool;
   //    Reset : Bool;
   //    REAC_DELAY { ExternalWritable := 'False'} : Time;
   //    Bypass_ET200 : Bool;
   // END_VAR
   // VAR_OUTPUT
   //    OUT_1 : Bool;
   //    OUT_2 : Bool;
   //    OUT_3 : Bool;
   //    OUT_4 : Bool;
   //    Diag_1 : Bool;
   //    Diag_2 : Bool;
   //    Diag_3 : Bool;
   //    Diag_4 : Bool;
   //    Lamp_1 : Bool;
   //    Lamp_2 : Bool;
   //    Lamp_3 : Bool;
   //    Lamp_4 : Bool;
   // END_VAR
   // VAR
   //    ESTOP_1 { S7_SetPoint := 'True'} : ESTOP1;
   //    ESTOP_2 { S7_SetPoint := 'True'} : ESTOP1;
   //    ESTOP_3 { S7_SetPoint := 'True'} : ESTOP1;
   //    ESTOP_4 { S7_SetPoint := 'True'} : ESTOP1;
   //    TON_1 { ExternalWritable := 'False'} : TON;
   //    TON_2 { ExternalWritable := 'False'} : TON;
   //    TON_3 { ExternalWritable := 'False'} : TON;
   //    TON_4 { ExternalWritable := 'False'} : TON;
   // END_VAR
BEGIN
END_DATA_BLOCK

DATA_BLOCK "n0046-ct1-el003-k30001_SN50_3"   // DB1038, F_DB
VERSION : 0.1
// stored: AutoNumber true, DBAccessibleFromOPCUA true, DBAccessibleFromWebserver true, InstanceOfName 00_Push-Button_Input, InstanceOfType FB
"00_Push-Button_Input"
   // VAR_INPUT
   //    IN_1 : Bool;
   //    IN_2 : Bool;
   //    IN_3 : Bool;
   //    IN_4 : Bool;
   //    ON_Tristate : Bool;
   //    ON_Lamp : Bool;
   //    Reset : Bool;
   //    REAC_DELAY { ExternalWritable := 'False'} : Time;
   //    Bypass_ET200 : Bool;
   // END_VAR
   // VAR_OUTPUT
   //    OUT_1 : Bool;
   //    OUT_2 : Bool;
   //    OUT_3 : Bool;
   //    OUT_4 : Bool;
   //    Diag_1 : Bool;
   //    Diag_2 : Bool;
   //    Diag_3 : Bool;
   //    Diag_4 : Bool;
   //    Lamp_1 : Bool;
   //    Lamp_2 : Bool;
   //    Lamp_3 : Bool;
   //    Lamp_4 : Bool;
   // END_VAR
   // VAR
   //    ESTOP_1 { S7_SetPoint := 'True'} : ESTOP1;
   //    ESTOP_2 { S7_SetPoint := 'True'} : ESTOP1;
   //    ESTOP_3 { S7_SetPoint := 'True'} : ESTOP1;
   //    ESTOP_4 { S7_SetPoint := 'True'} : ESTOP1;
   //    TON_1 { ExternalWritable := 'False'} : TON;
   //    TON_2 { ExternalWritable := 'False'} : TON;
   //    TON_3 { ExternalWritable := 'False'} : TON;
   //    TON_4 { ExternalWritable := 'False'} : TON;
   // END_VAR
BEGIN
END_DATA_BLOCK

DATA_BLOCK "n0046-ct1-el003-k30001_SN50_4"   // DB1039, F_DB
VERSION : 0.1
// stored: AutoNumber true, DBAccessibleFromOPCUA true, DBAccessibleFromWebserver true, InstanceOfName 00_Push-Button_Input, InstanceOfType FB
"00_Push-Button_Input"
   // VAR_INPUT
   //    IN_1 : Bool;
   //    IN_2 : Bool;
   //    IN_3 : Bool;
   //    IN_4 : Bool;
   //    ON_Tristate : Bool;
   //    ON_Lamp : Bool;
   //    Reset : Bool;
   //    REAC_DELAY { ExternalWritable := 'False'} : Time;
   //    Bypass_ET200 : Bool;
   // END_VAR
   // VAR_OUTPUT
   //    OUT_1 : Bool;
   //    OUT_2 : Bool;
   //    OUT_3 : Bool;
   //    OUT_4 : Bool;
   //    Diag_1 : Bool;
   //    Diag_2 : Bool;
   //    Diag_3 : Bool;
   //    Diag_4 : Bool;
   //    Lamp_1 : Bool;
   //    Lamp_2 : Bool;
   //    Lamp_3 : Bool;
   //    Lamp_4 : Bool;
   // END_VAR
   // VAR
   //    ESTOP_1 { S7_SetPoint := 'True'} : ESTOP1;
   //    ESTOP_2 { S7_SetPoint := 'True'} : ESTOP1;
   //    ESTOP_3 { S7_SetPoint := 'True'} : ESTOP1;
   //    ESTOP_4 { S7_SetPoint := 'True'} : ESTOP1;
   //    TON_1 { ExternalWritable := 'False'} : TON;
   //    TON_2 { ExternalWritable := 'False'} : TON;
   //    TON_3 { ExternalWritable := 'False'} : TON;
   //    TON_4 { ExternalWritable := 'False'} : TON;
   // END_VAR
BEGIN
END_DATA_BLOCK

DATA_BLOCK "n0050-uc13-el001-k30001_SN50_1"   // DB1040, F_DB
VERSION : 0.1
// stored: AutoNumber true, DBAccessibleFromOPCUA true, DBAccessibleFromWebserver true, InstanceOfName 00_Push-Button_Input, InstanceOfType FB
"00_Push-Button_Input"
   // VAR_INPUT
   //    IN_1 : Bool;
   //    IN_2 : Bool;
   //    IN_3 : Bool;
   //    IN_4 : Bool;
   //    ON_Tristate : Bool;
   //    ON_Lamp : Bool;
   //    Reset : Bool;
   //    REAC_DELAY { ExternalWritable := 'False'} : Time;
   //    Bypass_ET200 : Bool;
   // END_VAR
   // VAR_OUTPUT
   //    OUT_1 : Bool;
   //    OUT_2 : Bool;
   //    OUT_3 : Bool;
   //    OUT_4 : Bool;
   //    Diag_1 : Bool;
   //    Diag_2 : Bool;
   //    Diag_3 : Bool;
   //    Diag_4 : Bool;
   //    Lamp_1 : Bool;
   //    Lamp_2 : Bool;
   //    Lamp_3 : Bool;
   //    Lamp_4 : Bool;
   // END_VAR
   // VAR
   //    ESTOP_1 { S7_SetPoint := 'True'} : ESTOP1;
   //    ESTOP_2 { S7_SetPoint := 'True'} : ESTOP1;
   //    ESTOP_3 { S7_SetPoint := 'True'} : ESTOP1;
   //    ESTOP_4 { S7_SetPoint := 'True'} : ESTOP1;
   //    TON_1 { ExternalWritable := 'False'} : TON;
   //    TON_2 { ExternalWritable := 'False'} : TON;
   //    TON_3 { ExternalWritable := 'False'} : TON;
   //    TON_4 { ExternalWritable := 'False'} : TON;
   // END_VAR
BEGIN
END_DATA_BLOCK

DATA_BLOCK "n0050-uc13-el001-k30001_SN50_2"   // DB1041, F_DB
VERSION : 0.1
// stored: AutoNumber true, DBAccessibleFromOPCUA true, DBAccessibleFromWebserver true, InstanceOfName 00_Push-Button_Input, InstanceOfType FB
"00_Push-Button_Input"
   // VAR_INPUT
   //    IN_1 : Bool;
   //    IN_2 : Bool;
   //    IN_3 : Bool;
   //    IN_4 : Bool;
   //    ON_Tristate : Bool;
   //    ON_Lamp : Bool;
   //    Reset : Bool;
   //    REAC_DELAY { ExternalWritable := 'False'} : Time;
   //    Bypass_ET200 : Bool;
   // END_VAR
   // VAR_OUTPUT
   //    OUT_1 : Bool;
   //    OUT_2 : Bool;
   //    OUT_3 : Bool;
   //    OUT_4 : Bool;
   //    Diag_1 : Bool;
   //    Diag_2 : Bool;
   //    Diag_3 : Bool;
   //    Diag_4 : Bool;
   //    Lamp_1 : Bool;
   //    Lamp_2 : Bool;
   //    Lamp_3 : Bool;
   //    Lamp_4 : Bool;
   // END_VAR
   // VAR
   //    ESTOP_1 { S7_SetPoint := 'True'} : ESTOP1;
   //    ESTOP_2 { S7_SetPoint := 'True'} : ESTOP1;
   //    ESTOP_3 { S7_SetPoint := 'True'} : ESTOP1;
   //    ESTOP_4 { S7_SetPoint := 'True'} : ESTOP1;
   //    TON_1 { ExternalWritable := 'False'} : TON;
   //    TON_2 { ExternalWritable := 'False'} : TON;
   //    TON_3 { ExternalWritable := 'False'} : TON;
   //    TON_4 { ExternalWritable := 'False'} : TON;
   // END_VAR
BEGIN
END_DATA_BLOCK

DATA_BLOCK "n0050-uc13-el001-k30001_SN50_3"   // DB1042, F_DB
VERSION : 0.1
// stored: AutoNumber true, DBAccessibleFromOPCUA true, DBAccessibleFromWebserver true, InstanceOfName 00_Push-Button_Input, InstanceOfType FB
"00_Push-Button_Input"
   // VAR_INPUT
   //    IN_1 : Bool;
   //    IN_2 : Bool;
   //    IN_3 : Bool;
   //    IN_4 : Bool;
   //    ON_Tristate : Bool;
   //    ON_Lamp : Bool;
   //    Reset : Bool;
   //    REAC_DELAY { ExternalWritable := 'False'} : Time;
   //    Bypass_ET200 : Bool;
   // END_VAR
   // VAR_OUTPUT
   //    OUT_1 : Bool;
   //    OUT_2 : Bool;
   //    OUT_3 : Bool;
   //    OUT_4 : Bool;
   //    Diag_1 : Bool;
   //    Diag_2 : Bool;
   //    Diag_3 : Bool;
   //    Diag_4 : Bool;
   //    Lamp_1 : Bool;
   //    Lamp_2 : Bool;
   //    Lamp_3 : Bool;
   //    Lamp_4 : Bool;
   // END_VAR
   // VAR
   //    ESTOP_1 { S7_SetPoint := 'True'} : ESTOP1;
   //    ESTOP_2 { S7_SetPoint := 'True'} : ESTOP1;
   //    ESTOP_3 { S7_SetPoint := 'True'} : ESTOP1;
   //    ESTOP_4 { S7_SetPoint := 'True'} : ESTOP1;
   //    TON_1 { ExternalWritable := 'False'} : TON;
   //    TON_2 { ExternalWritable := 'False'} : TON;
   //    TON_3 { ExternalWritable := 'False'} : TON;
   //    TON_4 { ExternalWritable := 'False'} : TON;
   // END_VAR
BEGIN
END_DATA_BLOCK

DATA_BLOCK "n0051-uc134-xn10_SN50_1"   // DB1043, F_DB
VERSION : 0.1
// stored: AutoNumber true, DBAccessibleFromOPCUA true, DBAccessibleFromWebserver true, InstanceOfName 00_Push-Button_Input, InstanceOfType FB
"00_Push-Button_Input"
   // VAR_INPUT
   //    IN_1 : Bool;
   //    IN_2 : Bool;
   //    IN_3 : Bool;
   //    IN_4 : Bool;
   //    ON_Tristate : Bool;
   //    ON_Lamp : Bool;
   //    Reset : Bool;
   //    REAC_DELAY { ExternalWritable := 'False'} : Time;
   //    Bypass_ET200 : Bool;
   // END_VAR
   // VAR_OUTPUT
   //    OUT_1 : Bool;
   //    OUT_2 : Bool;
   //    OUT_3 : Bool;
   //    OUT_4 : Bool;
   //    Diag_1 : Bool;
   //    Diag_2 : Bool;
   //    Diag_3 : Bool;
   //    Diag_4 : Bool;
   //    Lamp_1 : Bool;
   //    Lamp_2 : Bool;
   //    Lamp_3 : Bool;
   //    Lamp_4 : Bool;
   // END_VAR
   // VAR
   //    ESTOP_1 { S7_SetPoint := 'True'} : ESTOP1;
   //    ESTOP_2 { S7_SetPoint := 'True'} : ESTOP1;
   //    ESTOP_3 { S7_SetPoint := 'True'} : ESTOP1;
   //    ESTOP_4 { S7_SetPoint := 'True'} : ESTOP1;
   //    TON_1 { ExternalWritable := 'False'} : TON;
   //    TON_2 { ExternalWritable := 'False'} : TON;
   //    TON_3 { ExternalWritable := 'False'} : TON;
   //    TON_4 { ExternalWritable := 'False'} : TON;
   // END_VAR
BEGIN
END_DATA_BLOCK

DATA_BLOCK "n0051-uc134-xn10_SN50_2"   // DB1044, F_DB
VERSION : 0.1
// stored: AutoNumber true, DBAccessibleFromOPCUA true, DBAccessibleFromWebserver true, InstanceOfName 00_Push-Button_Input, InstanceOfType FB
"00_Push-Button_Input"
   // VAR_INPUT
   //    IN_1 : Bool;
   //    IN_2 : Bool;
   //    IN_3 : Bool;
   //    IN_4 : Bool;
   //    ON_Tristate : Bool;
   //    ON_Lamp : Bool;
   //    Reset : Bool;
   //    REAC_DELAY { ExternalWritable := 'False'} : Time;
   //    Bypass_ET200 : Bool;
   // END_VAR
   // VAR_OUTPUT
   //    OUT_1 : Bool;
   //    OUT_2 : Bool;
   //    OUT_3 : Bool;
   //    OUT_4 : Bool;
   //    Diag_1 : Bool;
   //    Diag_2 : Bool;
   //    Diag_3 : Bool;
   //    Diag_4 : Bool;
   //    Lamp_1 : Bool;
   //    Lamp_2 : Bool;
   //    Lamp_3 : Bool;
   //    Lamp_4 : Bool;
   // END_VAR
   // VAR
   //    ESTOP_1 { S7_SetPoint := 'True'} : ESTOP1;
   //    ESTOP_2 { S7_SetPoint := 'True'} : ESTOP1;
   //    ESTOP_3 { S7_SetPoint := 'True'} : ESTOP1;
   //    ESTOP_4 { S7_SetPoint := 'True'} : ESTOP1;
   //    TON_1 { ExternalWritable := 'False'} : TON;
   //    TON_2 { ExternalWritable := 'False'} : TON;
   //    TON_3 { ExternalWritable := 'False'} : TON;
   //    TON_4 { ExternalWritable := 'False'} : TON;
   // END_VAR
BEGIN
END_DATA_BLOCK

DATA_BLOCK "n0053-uc12-el001-k30001_SN50_1"   // DB1045, F_DB
VERSION : 0.1
// stored: AutoNumber true, DBAccessibleFromOPCUA true, DBAccessibleFromWebserver true, InstanceOfName 00_Push-Button_Input, InstanceOfType FB
"00_Push-Button_Input"
   // VAR_INPUT
   //    IN_1 : Bool;
   //    IN_2 : Bool;
   //    IN_3 : Bool;
   //    IN_4 : Bool;
   //    ON_Tristate : Bool;
   //    ON_Lamp : Bool;
   //    Reset : Bool;
   //    REAC_DELAY { ExternalWritable := 'False'} : Time;
   //    Bypass_ET200 : Bool;
   // END_VAR
   // VAR_OUTPUT
   //    OUT_1 : Bool;
   //    OUT_2 : Bool;
   //    OUT_3 : Bool;
   //    OUT_4 : Bool;
   //    Diag_1 : Bool;
   //    Diag_2 : Bool;
   //    Diag_3 : Bool;
   //    Diag_4 : Bool;
   //    Lamp_1 : Bool;
   //    Lamp_2 : Bool;
   //    Lamp_3 : Bool;
   //    Lamp_4 : Bool;
   // END_VAR
   // VAR
   //    ESTOP_1 { S7_SetPoint := 'True'} : ESTOP1;
   //    ESTOP_2 { S7_SetPoint := 'True'} : ESTOP1;
   //    ESTOP_3 { S7_SetPoint := 'True'} : ESTOP1;
   //    ESTOP_4 { S7_SetPoint := 'True'} : ESTOP1;
   //    TON_1 { ExternalWritable := 'False'} : TON;
   //    TON_2 { ExternalWritable := 'False'} : TON;
   //    TON_3 { ExternalWritable := 'False'} : TON;
   //    TON_4 { ExternalWritable := 'False'} : TON;
   // END_VAR
BEGIN
END_DATA_BLOCK

DATA_BLOCK "n0053-uc12-el001-k30001_SN50_2"   // DB1046, F_DB
VERSION : 0.1
// stored: AutoNumber true, DBAccessibleFromOPCUA true, DBAccessibleFromWebserver true, InstanceOfName 00_Push-Button_Input, InstanceOfType FB
"00_Push-Button_Input"
   // VAR_INPUT
   //    IN_1 : Bool;
   //    IN_2 : Bool;
   //    IN_3 : Bool;
   //    IN_4 : Bool;
   //    ON_Tristate : Bool;
   //    ON_Lamp : Bool;
   //    Reset : Bool;
   //    REAC_DELAY { ExternalWritable := 'False'} : Time;
   //    Bypass_ET200 : Bool;
   // END_VAR
   // VAR_OUTPUT
   //    OUT_1 : Bool;
   //    OUT_2 : Bool;
   //    OUT_3 : Bool;
   //    OUT_4 : Bool;
   //    Diag_1 : Bool;
   //    Diag_2 : Bool;
   //    Diag_3 : Bool;
   //    Diag_4 : Bool;
   //    Lamp_1 : Bool;
   //    Lamp_2 : Bool;
   //    Lamp_3 : Bool;
   //    Lamp_4 : Bool;
   // END_VAR
   // VAR
   //    ESTOP_1 { S7_SetPoint := 'True'} : ESTOP1;
   //    ESTOP_2 { S7_SetPoint := 'True'} : ESTOP1;
   //    ESTOP_3 { S7_SetPoint := 'True'} : ESTOP1;
   //    ESTOP_4 { S7_SetPoint := 'True'} : ESTOP1;
   //    TON_1 { ExternalWritable := 'False'} : TON;
   //    TON_2 { ExternalWritable := 'False'} : TON;
   //    TON_3 { ExternalWritable := 'False'} : TON;
   //    TON_4 { ExternalWritable := 'False'} : TON;
   // END_VAR
BEGIN
END_DATA_BLOCK

DATA_BLOCK "n0053-uc12-el001-k30001_SN50_3"   // DB1047, F_DB
VERSION : 0.1
// stored: AutoNumber true, DBAccessibleFromOPCUA true, DBAccessibleFromWebserver true, InstanceOfName 00_Push-Button_Input, InstanceOfType FB
"00_Push-Button_Input"
   // VAR_INPUT
   //    IN_1 : Bool;
   //    IN_2 : Bool;
   //    IN_3 : Bool;
   //    IN_4 : Bool;
   //    ON_Tristate : Bool;
   //    ON_Lamp : Bool;
   //    Reset : Bool;
   //    REAC_DELAY { ExternalWritable := 'False'} : Time;
   //    Bypass_ET200 : Bool;
   // END_VAR
   // VAR_OUTPUT
   //    OUT_1 : Bool;
   //    OUT_2 : Bool;
   //    OUT_3 : Bool;
   //    OUT_4 : Bool;
   //    Diag_1 : Bool;
   //    Diag_2 : Bool;
   //    Diag_3 : Bool;
   //    Diag_4 : Bool;
   //    Lamp_1 : Bool;
   //    Lamp_2 : Bool;
   //    Lamp_3 : Bool;
   //    Lamp_4 : Bool;
   // END_VAR
   // VAR
   //    ESTOP_1 { S7_SetPoint := 'True'} : ESTOP1;
   //    ESTOP_2 { S7_SetPoint := 'True'} : ESTOP1;
   //    ESTOP_3 { S7_SetPoint := 'True'} : ESTOP1;
   //    ESTOP_4 { S7_SetPoint := 'True'} : ESTOP1;
   //    TON_1 { ExternalWritable := 'False'} : TON;
   //    TON_2 { ExternalWritable := 'False'} : TON;
   //    TON_3 { ExternalWritable := 'False'} : TON;
   //    TON_4 { ExternalWritable := 'False'} : TON;
   // END_VAR
BEGIN
END_DATA_BLOCK

DATA_BLOCK "n0055-uc124-xn10_SN50_1"   // DB1048, F_DB
VERSION : 0.1
// stored: AutoNumber true, DBAccessibleFromOPCUA true, DBAccessibleFromWebserver true, InstanceOfName 00_Push-Button_Input, InstanceOfType FB
"00_Push-Button_Input"
   // VAR_INPUT
   //    IN_1 : Bool;
   //    IN_2 : Bool;
   //    IN_3 : Bool;
   //    IN_4 : Bool;
   //    ON_Tristate : Bool;
   //    ON_Lamp : Bool;
   //    Reset : Bool;
   //    REAC_DELAY { ExternalWritable := 'False'} : Time;
   //    Bypass_ET200 : Bool;
   // END_VAR
   // VAR_OUTPUT
   //    OUT_1 : Bool;
   //    OUT_2 : Bool;
   //    OUT_3 : Bool;
   //    OUT_4 : Bool;
   //    Diag_1 : Bool;
   //    Diag_2 : Bool;
   //    Diag_3 : Bool;
   //    Diag_4 : Bool;
   //    Lamp_1 : Bool;
   //    Lamp_2 : Bool;
   //    Lamp_3 : Bool;
   //    Lamp_4 : Bool;
   // END_VAR
   // VAR
   //    ESTOP_1 { S7_SetPoint := 'True'} : ESTOP1;
   //    ESTOP_2 { S7_SetPoint := 'True'} : ESTOP1;
   //    ESTOP_3 { S7_SetPoint := 'True'} : ESTOP1;
   //    ESTOP_4 { S7_SetPoint := 'True'} : ESTOP1;
   //    TON_1 { ExternalWritable := 'False'} : TON;
   //    TON_2 { ExternalWritable := 'False'} : TON;
   //    TON_3 { ExternalWritable := 'False'} : TON;
   //    TON_4 { ExternalWritable := 'False'} : TON;
   // END_VAR
BEGIN
END_DATA_BLOCK

DATA_BLOCK "n0055-uc124-xn10_SN50_2"   // DB1049, F_DB
VERSION : 0.1
// stored: AutoNumber true, DBAccessibleFromOPCUA true, DBAccessibleFromWebserver true, InstanceOfName 00_Push-Button_Input, InstanceOfType FB
"00_Push-Button_Input"
   // VAR_INPUT
   //    IN_1 : Bool;
   //    IN_2 : Bool;
   //    IN_3 : Bool;
   //    IN_4 : Bool;
   //    ON_Tristate : Bool;
   //    ON_Lamp : Bool;
   //    Reset : Bool;
   //    REAC_DELAY { ExternalWritable := 'False'} : Time;
   //    Bypass_ET200 : Bool;
   // END_VAR
   // VAR_OUTPUT
   //    OUT_1 : Bool;
   //    OUT_2 : Bool;
   //    OUT_3 : Bool;
   //    OUT_4 : Bool;
   //    Diag_1 : Bool;
   //    Diag_2 : Bool;
   //    Diag_3 : Bool;
   //    Diag_4 : Bool;
   //    Lamp_1 : Bool;
   //    Lamp_2 : Bool;
   //    Lamp_3 : Bool;
   //    Lamp_4 : Bool;
   // END_VAR
   // VAR
   //    ESTOP_1 { S7_SetPoint := 'True'} : ESTOP1;
   //    ESTOP_2 { S7_SetPoint := 'True'} : ESTOP1;
   //    ESTOP_3 { S7_SetPoint := 'True'} : ESTOP1;
   //    ESTOP_4 { S7_SetPoint := 'True'} : ESTOP1;
   //    TON_1 { ExternalWritable := 'False'} : TON;
   //    TON_2 { ExternalWritable := 'False'} : TON;
   //    TON_3 { ExternalWritable := 'False'} : TON;
   //    TON_4 { ExternalWritable := 'False'} : TON;
   // END_VAR
BEGIN
END_DATA_BLOCK

DATA_BLOCK "n0057-uc11-el001-k30001_SN50_1"   // DB1050, F_DB
VERSION : 0.1
// stored: AutoNumber true, DBAccessibleFromOPCUA true, DBAccessibleFromWebserver true, InstanceOfName 00_Push-Button_Input, InstanceOfType FB
"00_Push-Button_Input"
   // VAR_INPUT
   //    IN_1 : Bool;
   //    IN_2 : Bool;
   //    IN_3 : Bool;
   //    IN_4 : Bool;
   //    ON_Tristate : Bool;
   //    ON_Lamp : Bool;
   //    Reset : Bool;
   //    REAC_DELAY { ExternalWritable := 'False'} : Time;
   //    Bypass_ET200 : Bool;
   // END_VAR
   // VAR_OUTPUT
   //    OUT_1 : Bool;
   //    OUT_2 : Bool;
   //    OUT_3 : Bool;
   //    OUT_4 : Bool;
   //    Diag_1 : Bool;
   //    Diag_2 : Bool;
   //    Diag_3 : Bool;
   //    Diag_4 : Bool;
   //    Lamp_1 : Bool;
   //    Lamp_2 : Bool;
   //    Lamp_3 : Bool;
   //    Lamp_4 : Bool;
   // END_VAR
   // VAR
   //    ESTOP_1 { S7_SetPoint := 'True'} : ESTOP1;
   //    ESTOP_2 { S7_SetPoint := 'True'} : ESTOP1;
   //    ESTOP_3 { S7_SetPoint := 'True'} : ESTOP1;
   //    ESTOP_4 { S7_SetPoint := 'True'} : ESTOP1;
   //    TON_1 { ExternalWritable := 'False'} : TON;
   //    TON_2 { ExternalWritable := 'False'} : TON;
   //    TON_3 { ExternalWritable := 'False'} : TON;
   //    TON_4 { ExternalWritable := 'False'} : TON;
   // END_VAR
BEGIN
END_DATA_BLOCK

DATA_BLOCK "n0057-uc11-el001-k30001_SN50_2"   // DB1051, F_DB
VERSION : 0.1
// stored: AutoNumber true, DBAccessibleFromOPCUA true, DBAccessibleFromWebserver true, InstanceOfName 00_Push-Button_Input, InstanceOfType FB
"00_Push-Button_Input"
   // VAR_INPUT
   //    IN_1 : Bool;
   //    IN_2 : Bool;
   //    IN_3 : Bool;
   //    IN_4 : Bool;
   //    ON_Tristate : Bool;
   //    ON_Lamp : Bool;
   //    Reset : Bool;
   //    REAC_DELAY { ExternalWritable := 'False'} : Time;
   //    Bypass_ET200 : Bool;
   // END_VAR
   // VAR_OUTPUT
   //    OUT_1 : Bool;
   //    OUT_2 : Bool;
   //    OUT_3 : Bool;
   //    OUT_4 : Bool;
   //    Diag_1 : Bool;
   //    Diag_2 : Bool;
   //    Diag_3 : Bool;
   //    Diag_4 : Bool;
   //    Lamp_1 : Bool;
   //    Lamp_2 : Bool;
   //    Lamp_3 : Bool;
   //    Lamp_4 : Bool;
   // END_VAR
   // VAR
   //    ESTOP_1 { S7_SetPoint := 'True'} : ESTOP1;
   //    ESTOP_2 { S7_SetPoint := 'True'} : ESTOP1;
   //    ESTOP_3 { S7_SetPoint := 'True'} : ESTOP1;
   //    ESTOP_4 { S7_SetPoint := 'True'} : ESTOP1;
   //    TON_1 { ExternalWritable := 'False'} : TON;
   //    TON_2 { ExternalWritable := 'False'} : TON;
   //    TON_3 { ExternalWritable := 'False'} : TON;
   //    TON_4 { ExternalWritable := 'False'} : TON;
   // END_VAR
BEGIN
END_DATA_BLOCK

DATA_BLOCK "n0057-uc11-el001-k30001_SN50_3"   // DB1052, F_DB
VERSION : 0.1
// stored: AutoNumber true, DBAccessibleFromOPCUA true, DBAccessibleFromWebserver true, InstanceOfName 00_Push-Button_Input, InstanceOfType FB
"00_Push-Button_Input"
   // VAR_INPUT
   //    IN_1 : Bool;
   //    IN_2 : Bool;
   //    IN_3 : Bool;
   //    IN_4 : Bool;
   //    ON_Tristate : Bool;
   //    ON_Lamp : Bool;
   //    Reset : Bool;
   //    REAC_DELAY { ExternalWritable := 'False'} : Time;
   //    Bypass_ET200 : Bool;
   // END_VAR
   // VAR_OUTPUT
   //    OUT_1 : Bool;
   //    OUT_2 : Bool;
   //    OUT_3 : Bool;
   //    OUT_4 : Bool;
   //    Diag_1 : Bool;
   //    Diag_2 : Bool;
   //    Diag_3 : Bool;
   //    Diag_4 : Bool;
   //    Lamp_1 : Bool;
   //    Lamp_2 : Bool;
   //    Lamp_3 : Bool;
   //    Lamp_4 : Bool;
   // END_VAR
   // VAR
   //    ESTOP_1 { S7_SetPoint := 'True'} : ESTOP1;
   //    ESTOP_2 { S7_SetPoint := 'True'} : ESTOP1;
   //    ESTOP_3 { S7_SetPoint := 'True'} : ESTOP1;
   //    ESTOP_4 { S7_SetPoint := 'True'} : ESTOP1;
   //    TON_1 { ExternalWritable := 'False'} : TON;
   //    TON_2 { ExternalWritable := 'False'} : TON;
   //    TON_3 { ExternalWritable := 'False'} : TON;
   //    TON_4 { ExternalWritable := 'False'} : TON;
   // END_VAR
BEGIN
END_DATA_BLOCK

DATA_BLOCK "n0060-uc114-xn10_SN50_1"   // DB1053, F_DB
VERSION : 0.1
// stored: AutoNumber true, DBAccessibleFromOPCUA true, DBAccessibleFromWebserver true, InstanceOfName 00_Push-Button_Input, InstanceOfType FB
"00_Push-Button_Input"
   // VAR_INPUT
   //    IN_1 : Bool;
   //    IN_2 : Bool;
   //    IN_3 : Bool;
   //    IN_4 : Bool;
   //    ON_Tristate : Bool;
   //    ON_Lamp : Bool;
   //    Reset : Bool;
   //    REAC_DELAY { ExternalWritable := 'False'} : Time;
   //    Bypass_ET200 : Bool;
   // END_VAR
   // VAR_OUTPUT
   //    OUT_1 : Bool;
   //    OUT_2 : Bool;
   //    OUT_3 : Bool;
   //    OUT_4 : Bool;
   //    Diag_1 : Bool;
   //    Diag_2 : Bool;
   //    Diag_3 : Bool;
   //    Diag_4 : Bool;
   //    Lamp_1 : Bool;
   //    Lamp_2 : Bool;
   //    Lamp_3 : Bool;
   //    Lamp_4 : Bool;
   // END_VAR
   // VAR
   //    ESTOP_1 { S7_SetPoint := 'True'} : ESTOP1;
   //    ESTOP_2 { S7_SetPoint := 'True'} : ESTOP1;
   //    ESTOP_3 { S7_SetPoint := 'True'} : ESTOP1;
   //    ESTOP_4 { S7_SetPoint := 'True'} : ESTOP1;
   //    TON_1 { ExternalWritable := 'False'} : TON;
   //    TON_2 { ExternalWritable := 'False'} : TON;
   //    TON_3 { ExternalWritable := 'False'} : TON;
   //    TON_4 { ExternalWritable := 'False'} : TON;
   // END_VAR
BEGIN
END_DATA_BLOCK

DATA_BLOCK "n0060-uc114-xn10_SN50_2"   // DB1054, F_DB
VERSION : 0.1
// stored: AutoNumber true, DBAccessibleFromOPCUA true, DBAccessibleFromWebserver true, InstanceOfName 00_Push-Button_Input, InstanceOfType FB
"00_Push-Button_Input"
   // VAR_INPUT
   //    IN_1 : Bool;
   //    IN_2 : Bool;
   //    IN_3 : Bool;
   //    IN_4 : Bool;
   //    ON_Tristate : Bool;
   //    ON_Lamp : Bool;
   //    Reset : Bool;
   //    REAC_DELAY { ExternalWritable := 'False'} : Time;
   //    Bypass_ET200 : Bool;
   // END_VAR
   // VAR_OUTPUT
   //    OUT_1 : Bool;
   //    OUT_2 : Bool;
   //    OUT_3 : Bool;
   //    OUT_4 : Bool;
   //    Diag_1 : Bool;
   //    Diag_2 : Bool;
   //    Diag_3 : Bool;
   //    Diag_4 : Bool;
   //    Lamp_1 : Bool;
   //    Lamp_2 : Bool;
   //    Lamp_3 : Bool;
   //    Lamp_4 : Bool;
   // END_VAR
   // VAR
   //    ESTOP_1 { S7_SetPoint := 'True'} : ESTOP1;
   //    ESTOP_2 { S7_SetPoint := 'True'} : ESTOP1;
   //    ESTOP_3 { S7_SetPoint := 'True'} : ESTOP1;
   //    ESTOP_4 { S7_SetPoint := 'True'} : ESTOP1;
   //    TON_1 { ExternalWritable := 'False'} : TON;
   //    TON_2 { ExternalWritable := 'False'} : TON;
   //    TON_3 { ExternalWritable := 'False'} : TON;
   //    TON_4 { ExternalWritable := 'False'} : TON;
   // END_VAR
BEGIN
END_DATA_BLOCK

DATA_BLOCK "n0028-uc17-el001-k30001_SN50_1"   // DB1055, F_DB
VERSION : 0.1
// stored: AutoNumber true, DBAccessibleFromOPCUA true, DBAccessibleFromWebserver true, InstanceOfName 00_Push-Button_Input, InstanceOfType FB
"00_Push-Button_Input"
   // VAR_INPUT
   //    IN_1 : Bool;
   //    IN_2 : Bool;
   //    IN_3 : Bool;
   //    IN_4 : Bool;
   //    ON_Tristate : Bool;
   //    ON_Lamp : Bool;
   //    Reset : Bool;
   //    REAC_DELAY { ExternalWritable := 'False'} : Time;
   //    Bypass_ET200 : Bool;
   // END_VAR
   // VAR_OUTPUT
   //    OUT_1 : Bool;
   //    OUT_2 : Bool;
   //    OUT_3 : Bool;
   //    OUT_4 : Bool;
   //    Diag_1 : Bool;
   //    Diag_2 : Bool;
   //    Diag_3 : Bool;
   //    Diag_4 : Bool;
   //    Lamp_1 : Bool;
   //    Lamp_2 : Bool;
   //    Lamp_3 : Bool;
   //    Lamp_4 : Bool;
   // END_VAR
   // VAR
   //    ESTOP_1 { S7_SetPoint := 'True'} : ESTOP1;
   //    ESTOP_2 { S7_SetPoint := 'True'} : ESTOP1;
   //    ESTOP_3 { S7_SetPoint := 'True'} : ESTOP1;
   //    ESTOP_4 { S7_SetPoint := 'True'} : ESTOP1;
   //    TON_1 { ExternalWritable := 'False'} : TON;
   //    TON_2 { ExternalWritable := 'False'} : TON;
   //    TON_3 { ExternalWritable := 'False'} : TON;
   //    TON_4 { ExternalWritable := 'False'} : TON;
   // END_VAR
BEGIN
END_DATA_BLOCK

DATA_BLOCK "n0028-uc17-el001-k30001_SN50_2"   // DB1056, F_DB
VERSION : 0.1
// stored: AutoNumber true, DBAccessibleFromOPCUA true, DBAccessibleFromWebserver true, InstanceOfName 00_Push-Button_Input, InstanceOfType FB
"00_Push-Button_Input"
   // VAR_INPUT
   //    IN_1 : Bool;
   //    IN_2 : Bool;
   //    IN_3 : Bool;
   //    IN_4 : Bool;
   //    ON_Tristate : Bool;
   //    ON_Lamp : Bool;
   //    Reset : Bool;
   //    REAC_DELAY { ExternalWritable := 'False'} : Time;
   //    Bypass_ET200 : Bool;
   // END_VAR
   // VAR_OUTPUT
   //    OUT_1 : Bool;
   //    OUT_2 : Bool;
   //    OUT_3 : Bool;
   //    OUT_4 : Bool;
   //    Diag_1 : Bool;
   //    Diag_2 : Bool;
   //    Diag_3 : Bool;
   //    Diag_4 : Bool;
   //    Lamp_1 : Bool;
   //    Lamp_2 : Bool;
   //    Lamp_3 : Bool;
   //    Lamp_4 : Bool;
   // END_VAR
   // VAR
   //    ESTOP_1 { S7_SetPoint := 'True'} : ESTOP1;
   //    ESTOP_2 { S7_SetPoint := 'True'} : ESTOP1;
   //    ESTOP_3 { S7_SetPoint := 'True'} : ESTOP1;
   //    ESTOP_4 { S7_SetPoint := 'True'} : ESTOP1;
   //    TON_1 { ExternalWritable := 'False'} : TON;
   //    TON_2 { ExternalWritable := 'False'} : TON;
   //    TON_3 { ExternalWritable := 'False'} : TON;
   //    TON_4 { ExternalWritable := 'False'} : TON;
   // END_VAR
BEGIN
END_DATA_BLOCK

DATA_BLOCK "n0029-uc173-xn10_SN50_1"   // DB1057, F_DB
VERSION : 0.1
// stored: AutoNumber true, DBAccessibleFromOPCUA true, DBAccessibleFromWebserver true, InstanceOfName 00_Push-Button_Input, InstanceOfType FB
"00_Push-Button_Input"
   // VAR_INPUT
   //    IN_1 : Bool;
   //    IN_2 : Bool;
   //    IN_3 : Bool;
   //    IN_4 : Bool;
   //    ON_Tristate : Bool;
   //    ON_Lamp : Bool;
   //    Reset : Bool;
   //    REAC_DELAY { ExternalWritable := 'False'} : Time;
   //    Bypass_ET200 : Bool;
   // END_VAR
   // VAR_OUTPUT
   //    OUT_1 : Bool;
   //    OUT_2 : Bool;
   //    OUT_3 : Bool;
   //    OUT_4 : Bool;
   //    Diag_1 : Bool;
   //    Diag_2 : Bool;
   //    Diag_3 : Bool;
   //    Diag_4 : Bool;
   //    Lamp_1 : Bool;
   //    Lamp_2 : Bool;
   //    Lamp_3 : Bool;
   //    Lamp_4 : Bool;
   // END_VAR
   // VAR
   //    ESTOP_1 { S7_SetPoint := 'True'} : ESTOP1;
   //    ESTOP_2 { S7_SetPoint := 'True'} : ESTOP1;
   //    ESTOP_3 { S7_SetPoint := 'True'} : ESTOP1;
   //    ESTOP_4 { S7_SetPoint := 'True'} : ESTOP1;
   //    TON_1 { ExternalWritable := 'False'} : TON;
   //    TON_2 { ExternalWritable := 'False'} : TON;
   //    TON_3 { ExternalWritable := 'False'} : TON;
   //    TON_4 { ExternalWritable := 'False'} : TON;
   // END_VAR
BEGIN
END_DATA_BLOCK

DATA_BLOCK "n0029-uc173-xn10_SN50_2"   // DB1058, F_DB
VERSION : 0.1
// stored: AutoNumber true, DBAccessibleFromOPCUA true, DBAccessibleFromWebserver true, InstanceOfName 00_Push-Button_Input, InstanceOfType FB
"00_Push-Button_Input"
   // VAR_INPUT
   //    IN_1 : Bool;
   //    IN_2 : Bool;
   //    IN_3 : Bool;
   //    IN_4 : Bool;
   //    ON_Tristate : Bool;
   //    ON_Lamp : Bool;
   //    Reset : Bool;
   //    REAC_DELAY { ExternalWritable := 'False'} : Time;
   //    Bypass_ET200 : Bool;
   // END_VAR
   // VAR_OUTPUT
   //    OUT_1 : Bool;
   //    OUT_2 : Bool;
   //    OUT_3 : Bool;
   //    OUT_4 : Bool;
   //    Diag_1 : Bool;
   //    Diag_2 : Bool;
   //    Diag_3 : Bool;
   //    Diag_4 : Bool;
   //    Lamp_1 : Bool;
   //    Lamp_2 : Bool;
   //    Lamp_3 : Bool;
   //    Lamp_4 : Bool;
   // END_VAR
   // VAR
   //    ESTOP_1 { S7_SetPoint := 'True'} : ESTOP1;
   //    ESTOP_2 { S7_SetPoint := 'True'} : ESTOP1;
   //    ESTOP_3 { S7_SetPoint := 'True'} : ESTOP1;
   //    ESTOP_4 { S7_SetPoint := 'True'} : ESTOP1;
   //    TON_1 { ExternalWritable := 'False'} : TON;
   //    TON_2 { ExternalWritable := 'False'} : TON;
   //    TON_3 { ExternalWritable := 'False'} : TON;
   //    TON_4 { ExternalWritable := 'False'} : TON;
   // END_VAR
BEGIN
END_DATA_BLOCK

DATA_BLOCK "n0033-zp001-el001-k40001_SN50_1"   // DB1059, F_DB
VERSION : 0.1
// stored: AutoNumber true, DBAccessibleFromOPCUA true, DBAccessibleFromWebserver true, InstanceOfName 00_Push-Button_Input, InstanceOfType FB
"00_Push-Button_Input"
   // VAR_INPUT
   //    IN_1 : Bool;
   //    IN_2 : Bool;
   //    IN_3 : Bool;
   //    IN_4 : Bool;
   //    ON_Tristate : Bool;
   //    ON_Lamp : Bool;
   //    Reset : Bool;
   //    REAC_DELAY { ExternalWritable := 'False'} : Time;
   //    Bypass_ET200 : Bool;
   // END_VAR
   // VAR_OUTPUT
   //    OUT_1 : Bool;
   //    OUT_2 : Bool;
   //    OUT_3 : Bool;
   //    OUT_4 : Bool;
   //    Diag_1 : Bool;
   //    Diag_2 : Bool;
   //    Diag_3 : Bool;
   //    Diag_4 : Bool;
   //    Lamp_1 : Bool;
   //    Lamp_2 : Bool;
   //    Lamp_3 : Bool;
   //    Lamp_4 : Bool;
   // END_VAR
   // VAR
   //    ESTOP_1 { S7_SetPoint := 'True'} : ESTOP1;
   //    ESTOP_2 { S7_SetPoint := 'True'} : ESTOP1;
   //    ESTOP_3 { S7_SetPoint := 'True'} : ESTOP1;
   //    ESTOP_4 { S7_SetPoint := 'True'} : ESTOP1;
   //    TON_1 { ExternalWritable := 'False'} : TON;
   //    TON_2 { ExternalWritable := 'False'} : TON;
   //    TON_3 { ExternalWritable := 'False'} : TON;
   //    TON_4 { ExternalWritable := 'False'} : TON;
   // END_VAR
BEGIN
END_DATA_BLOCK

DATA_BLOCK "n0033-zp001-el001-k40001_SN50_2"   // DB1060, F_DB
VERSION : 0.1
// stored: AutoNumber true, DBAccessibleFromOPCUA true, DBAccessibleFromWebserver true, InstanceOfName 00_Push-Button_Input, InstanceOfType FB
"00_Push-Button_Input"
   // VAR_INPUT
   //    IN_1 : Bool;
   //    IN_2 : Bool;
   //    IN_3 : Bool;
   //    IN_4 : Bool;
   //    ON_Tristate : Bool;
   //    ON_Lamp : Bool;
   //    Reset : Bool;
   //    REAC_DELAY { ExternalWritable := 'False'} : Time;
   //    Bypass_ET200 : Bool;
   // END_VAR
   // VAR_OUTPUT
   //    OUT_1 : Bool;
   //    OUT_2 : Bool;
   //    OUT_3 : Bool;
   //    OUT_4 : Bool;
   //    Diag_1 : Bool;
   //    Diag_2 : Bool;
   //    Diag_3 : Bool;
   //    Diag_4 : Bool;
   //    Lamp_1 : Bool;
   //    Lamp_2 : Bool;
   //    Lamp_3 : Bool;
   //    Lamp_4 : Bool;
   // END_VAR
   // VAR
   //    ESTOP_1 { S7_SetPoint := 'True'} : ESTOP1;
   //    ESTOP_2 { S7_SetPoint := 'True'} : ESTOP1;
   //    ESTOP_3 { S7_SetPoint := 'True'} : ESTOP1;
   //    ESTOP_4 { S7_SetPoint := 'True'} : ESTOP1;
   //    TON_1 { ExternalWritable := 'False'} : TON;
   //    TON_2 { ExternalWritable := 'False'} : TON;
   //    TON_3 { ExternalWritable := 'False'} : TON;
   //    TON_4 { ExternalWritable := 'False'} : TON;
   // END_VAR
BEGIN
END_DATA_BLOCK

DATA_BLOCK "n0033-zp001-el001-k40001_SN50_3"   // DB1061, F_DB
VERSION : 0.1
// stored: AutoNumber true, DBAccessibleFromOPCUA true, DBAccessibleFromWebserver true, InstanceOfName 00_Push-Button_Input, InstanceOfType FB
"00_Push-Button_Input"
   // VAR_INPUT
   //    IN_1 : Bool;
   //    IN_2 : Bool;
   //    IN_3 : Bool;
   //    IN_4 : Bool;
   //    ON_Tristate : Bool;
   //    ON_Lamp : Bool;
   //    Reset : Bool;
   //    REAC_DELAY { ExternalWritable := 'False'} : Time;
   //    Bypass_ET200 : Bool;
   // END_VAR
   // VAR_OUTPUT
   //    OUT_1 : Bool;
   //    OUT_2 : Bool;
   //    OUT_3 : Bool;
   //    OUT_4 : Bool;
   //    Diag_1 : Bool;
   //    Diag_2 : Bool;
   //    Diag_3 : Bool;
   //    Diag_4 : Bool;
   //    Lamp_1 : Bool;
   //    Lamp_2 : Bool;
   //    Lamp_3 : Bool;
   //    Lamp_4 : Bool;
   // END_VAR
   // VAR
   //    ESTOP_1 { S7_SetPoint := 'True'} : ESTOP1;
   //    ESTOP_2 { S7_SetPoint := 'True'} : ESTOP1;
   //    ESTOP_3 { S7_SetPoint := 'True'} : ESTOP1;
   //    ESTOP_4 { S7_SetPoint := 'True'} : ESTOP1;
   //    TON_1 { ExternalWritable := 'False'} : TON;
   //    TON_2 { ExternalWritable := 'False'} : TON;
   //    TON_3 { ExternalWritable := 'False'} : TON;
   //    TON_4 { ExternalWritable := 'False'} : TON;
   // END_VAR
BEGIN
END_DATA_BLOCK

DATA_BLOCK "n0034-ug6-el001-k30001_SN50_1"   // DB1062, F_DB
VERSION : 0.1
// stored: AutoNumber true, DBAccessibleFromOPCUA true, DBAccessibleFromWebserver true, InstanceOfName 00_Push-Button_Input, InstanceOfType FB
"00_Push-Button_Input"
   // VAR_INPUT
   //    IN_1 : Bool;
   //    IN_2 : Bool;
   //    IN_3 : Bool;
   //    IN_4 : Bool;
   //    ON_Tristate : Bool;
   //    ON_Lamp : Bool;
   //    Reset : Bool;
   //    REAC_DELAY { ExternalWritable := 'False'} : Time;
   //    Bypass_ET200 : Bool;
   // END_VAR
   // VAR_OUTPUT
   //    OUT_1 : Bool;
   //    OUT_2 : Bool;
   //    OUT_3 : Bool;
   //    OUT_4 : Bool;
   //    Diag_1 : Bool;
   //    Diag_2 : Bool;
   //    Diag_3 : Bool;
   //    Diag_4 : Bool;
   //    Lamp_1 : Bool;
   //    Lamp_2 : Bool;
   //    Lamp_3 : Bool;
   //    Lamp_4 : Bool;
   // END_VAR
   // VAR
   //    ESTOP_1 { S7_SetPoint := 'True'} : ESTOP1;
   //    ESTOP_2 { S7_SetPoint := 'True'} : ESTOP1;
   //    ESTOP_3 { S7_SetPoint := 'True'} : ESTOP1;
   //    ESTOP_4 { S7_SetPoint := 'True'} : ESTOP1;
   //    TON_1 { ExternalWritable := 'False'} : TON;
   //    TON_2 { ExternalWritable := 'False'} : TON;
   //    TON_3 { ExternalWritable := 'False'} : TON;
   //    TON_4 { ExternalWritable := 'False'} : TON;
   // END_VAR
BEGIN
END_DATA_BLOCK

DATA_BLOCK "n0034-ug6-el001-k30001_SN50_2"   // DB1063, F_DB
VERSION : 0.1
// stored: AutoNumber true, DBAccessibleFromOPCUA true, DBAccessibleFromWebserver true, InstanceOfName 00_Push-Button_Input, InstanceOfType FB
"00_Push-Button_Input"
   // VAR_INPUT
   //    IN_1 : Bool;
   //    IN_2 : Bool;
   //    IN_3 : Bool;
   //    IN_4 : Bool;
   //    ON_Tristate : Bool;
   //    ON_Lamp : Bool;
   //    Reset : Bool;
   //    REAC_DELAY { ExternalWritable := 'False'} : Time;
   //    Bypass_ET200 : Bool;
   // END_VAR
   // VAR_OUTPUT
   //    OUT_1 : Bool;
   //    OUT_2 : Bool;
   //    OUT_3 : Bool;
   //    OUT_4 : Bool;
   //    Diag_1 : Bool;
   //    Diag_2 : Bool;
   //    Diag_3 : Bool;
   //    Diag_4 : Bool;
   //    Lamp_1 : Bool;
   //    Lamp_2 : Bool;
   //    Lamp_3 : Bool;
   //    Lamp_4 : Bool;
   // END_VAR
   // VAR
   //    ESTOP_1 { S7_SetPoint := 'True'} : ESTOP1;
   //    ESTOP_2 { S7_SetPoint := 'True'} : ESTOP1;
   //    ESTOP_3 { S7_SetPoint := 'True'} : ESTOP1;
   //    ESTOP_4 { S7_SetPoint := 'True'} : ESTOP1;
   //    TON_1 { ExternalWritable := 'False'} : TON;
   //    TON_2 { ExternalWritable := 'False'} : TON;
   //    TON_3 { ExternalWritable := 'False'} : TON;
   //    TON_4 { ExternalWritable := 'False'} : TON;
   // END_VAR
BEGIN
END_DATA_BLOCK

DATA_BLOCK "n0034-ug6-el001-k30001_SN50_3"   // DB1064, F_DB
VERSION : 0.1
// stored: AutoNumber true, DBAccessibleFromOPCUA true, DBAccessibleFromWebserver true, InstanceOfName 00_Push-Button_Input, InstanceOfType FB
"00_Push-Button_Input"
   // VAR_INPUT
   //    IN_1 : Bool;
   //    IN_2 : Bool;
   //    IN_3 : Bool;
   //    IN_4 : Bool;
   //    ON_Tristate : Bool;
   //    ON_Lamp : Bool;
   //    Reset : Bool;
   //    REAC_DELAY { ExternalWritable := 'False'} : Time;
   //    Bypass_ET200 : Bool;
   // END_VAR
   // VAR_OUTPUT
   //    OUT_1 : Bool;
   //    OUT_2 : Bool;
   //    OUT_3 : Bool;
   //    OUT_4 : Bool;
   //    Diag_1 : Bool;
   //    Diag_2 : Bool;
   //    Diag_3 : Bool;
   //    Diag_4 : Bool;
   //    Lamp_1 : Bool;
   //    Lamp_2 : Bool;
   //    Lamp_3 : Bool;
   //    Lamp_4 : Bool;
   // END_VAR
   // VAR
   //    ESTOP_1 { S7_SetPoint := 'True'} : ESTOP1;
   //    ESTOP_2 { S7_SetPoint := 'True'} : ESTOP1;
   //    ESTOP_3 { S7_SetPoint := 'True'} : ESTOP1;
   //    ESTOP_4 { S7_SetPoint := 'True'} : ESTOP1;
   //    TON_1 { ExternalWritable := 'False'} : TON;
   //    TON_2 { ExternalWritable := 'False'} : TON;
   //    TON_3 { ExternalWritable := 'False'} : TON;
   //    TON_4 { ExternalWritable := 'False'} : TON;
   // END_VAR
BEGIN
END_DATA_BLOCK

DATA_BLOCK "n0035-ug6-xn10_SN50_1"   // DB1065, F_DB
VERSION : 0.1
// stored: AutoNumber true, DBAccessibleFromOPCUA true, DBAccessibleFromWebserver true, InstanceOfName 00_Push-Button_Input, InstanceOfType FB
"00_Push-Button_Input"
   // VAR_INPUT
   //    IN_1 : Bool;
   //    IN_2 : Bool;
   //    IN_3 : Bool;
   //    IN_4 : Bool;
   //    ON_Tristate : Bool;
   //    ON_Lamp : Bool;
   //    Reset : Bool;
   //    REAC_DELAY { ExternalWritable := 'False'} : Time;
   //    Bypass_ET200 : Bool;
   // END_VAR
   // VAR_OUTPUT
   //    OUT_1 : Bool;
   //    OUT_2 : Bool;
   //    OUT_3 : Bool;
   //    OUT_4 : Bool;
   //    Diag_1 : Bool;
   //    Diag_2 : Bool;
   //    Diag_3 : Bool;
   //    Diag_4 : Bool;
   //    Lamp_1 : Bool;
   //    Lamp_2 : Bool;
   //    Lamp_3 : Bool;
   //    Lamp_4 : Bool;
   // END_VAR
   // VAR
   //    ESTOP_1 { S7_SetPoint := 'True'} : ESTOP1;
   //    ESTOP_2 { S7_SetPoint := 'True'} : ESTOP1;
   //    ESTOP_3 { S7_SetPoint := 'True'} : ESTOP1;
   //    ESTOP_4 { S7_SetPoint := 'True'} : ESTOP1;
   //    TON_1 { ExternalWritable := 'False'} : TON;
   //    TON_2 { ExternalWritable := 'False'} : TON;
   //    TON_3 { ExternalWritable := 'False'} : TON;
   //    TON_4 { ExternalWritable := 'False'} : TON;
   // END_VAR
BEGIN
END_DATA_BLOCK

DATA_BLOCK "n0035-ug6-xn10_SN50_2"   // DB1066, F_DB
VERSION : 0.1
// stored: AutoNumber true, DBAccessibleFromOPCUA true, DBAccessibleFromWebserver true, InstanceOfName 00_Push-Button_Input, InstanceOfType FB
"00_Push-Button_Input"
   // VAR_INPUT
   //    IN_1 : Bool;
   //    IN_2 : Bool;
   //    IN_3 : Bool;
   //    IN_4 : Bool;
   //    ON_Tristate : Bool;
   //    ON_Lamp : Bool;
   //    Reset : Bool;
   //    REAC_DELAY { ExternalWritable := 'False'} : Time;
   //    Bypass_ET200 : Bool;
   // END_VAR
   // VAR_OUTPUT
   //    OUT_1 : Bool;
   //    OUT_2 : Bool;
   //    OUT_3 : Bool;
   //    OUT_4 : Bool;
   //    Diag_1 : Bool;
   //    Diag_2 : Bool;
   //    Diag_3 : Bool;
   //    Diag_4 : Bool;
   //    Lamp_1 : Bool;
   //    Lamp_2 : Bool;
   //    Lamp_3 : Bool;
   //    Lamp_4 : Bool;
   // END_VAR
   // VAR
   //    ESTOP_1 { S7_SetPoint := 'True'} : ESTOP1;
   //    ESTOP_2 { S7_SetPoint := 'True'} : ESTOP1;
   //    ESTOP_3 { S7_SetPoint := 'True'} : ESTOP1;
   //    ESTOP_4 { S7_SetPoint := 'True'} : ESTOP1;
   //    TON_1 { ExternalWritable := 'False'} : TON;
   //    TON_2 { ExternalWritable := 'False'} : TON;
   //    TON_3 { ExternalWritable := 'False'} : TON;
   //    TON_4 { ExternalWritable := 'False'} : TON;
   // END_VAR
BEGIN
END_DATA_BLOCK

DATA_BLOCK "n0043-db93-el001-k30001_SN50_1"   // DB1067, F_DB
VERSION : 0.1
// stored: AutoNumber true, DBAccessibleFromOPCUA true, DBAccessibleFromWebserver true, InstanceOfName 00_Push-Button_Input, InstanceOfType FB
"00_Push-Button_Input"
   // VAR_INPUT
   //    IN_1 : Bool;
   //    IN_2 : Bool;
   //    IN_3 : Bool;
   //    IN_4 : Bool;
   //    ON_Tristate : Bool;
   //    ON_Lamp : Bool;
   //    Reset : Bool;
   //    REAC_DELAY { ExternalWritable := 'False'} : Time;
   //    Bypass_ET200 : Bool;
   // END_VAR
   // VAR_OUTPUT
   //    OUT_1 : Bool;
   //    OUT_2 : Bool;
   //    OUT_3 : Bool;
   //    OUT_4 : Bool;
   //    Diag_1 : Bool;
   //    Diag_2 : Bool;
   //    Diag_3 : Bool;
   //    Diag_4 : Bool;
   //    Lamp_1 : Bool;
   //    Lamp_2 : Bool;
   //    Lamp_3 : Bool;
   //    Lamp_4 : Bool;
   // END_VAR
   // VAR
   //    ESTOP_1 { S7_SetPoint := 'True'} : ESTOP1;
   //    ESTOP_2 { S7_SetPoint := 'True'} : ESTOP1;
   //    ESTOP_3 { S7_SetPoint := 'True'} : ESTOP1;
   //    ESTOP_4 { S7_SetPoint := 'True'} : ESTOP1;
   //    TON_1 { ExternalWritable := 'False'} : TON;
   //    TON_2 { ExternalWritable := 'False'} : TON;
   //    TON_3 { ExternalWritable := 'False'} : TON;
   //    TON_4 { ExternalWritable := 'False'} : TON;
   // END_VAR
BEGIN
END_DATA_BLOCK

DATA_BLOCK "n0031-db931-xn10_SN50_1"   // DB1068, F_DB
VERSION : 0.1
// stored: AutoNumber true, DBAccessibleFromOPCUA true, DBAccessibleFromWebserver true, InstanceOfName 00_Push-Button_Input, InstanceOfType FB
"00_Push-Button_Input"
   // VAR_INPUT
   //    IN_1 : Bool;
   //    IN_2 : Bool;
   //    IN_3 : Bool;
   //    IN_4 : Bool;
   //    ON_Tristate : Bool;
   //    ON_Lamp : Bool;
   //    Reset : Bool;
   //    REAC_DELAY { ExternalWritable := 'False'} : Time;
   //    Bypass_ET200 : Bool;
   // END_VAR
   // VAR_OUTPUT
   //    OUT_1 : Bool;
   //    OUT_2 : Bool;
   //    OUT_3 : Bool;
   //    OUT_4 : Bool;
   //    Diag_1 : Bool;
   //    Diag_2 : Bool;
   //    Diag_3 : Bool;
   //    Diag_4 : Bool;
   //    Lamp_1 : Bool;
   //    Lamp_2 : Bool;
   //    Lamp_3 : Bool;
   //    Lamp_4 : Bool;
   // END_VAR
   // VAR
   //    ESTOP_1 { S7_SetPoint := 'True'} : ESTOP1;
   //    ESTOP_2 { S7_SetPoint := 'True'} : ESTOP1;
   //    ESTOP_3 { S7_SetPoint := 'True'} : ESTOP1;
   //    ESTOP_4 { S7_SetPoint := 'True'} : ESTOP1;
   //    TON_1 { ExternalWritable := 'False'} : TON;
   //    TON_2 { ExternalWritable := 'False'} : TON;
   //    TON_3 { ExternalWritable := 'False'} : TON;
   //    TON_4 { ExternalWritable := 'False'} : TON;
   // END_VAR
BEGIN
END_DATA_BLOCK

DATA_BLOCK "n0031-db931-xn10_SN50_2"   // DB1069, F_DB
VERSION : 0.1
// stored: AutoNumber true, DBAccessibleFromOPCUA true, DBAccessibleFromWebserver true, InstanceOfName 00_Push-Button_Input, InstanceOfType FB
"00_Push-Button_Input"
   // VAR_INPUT
   //    IN_1 : Bool;
   //    IN_2 : Bool;
   //    IN_3 : Bool;
   //    IN_4 : Bool;
   //    ON_Tristate : Bool;
   //    ON_Lamp : Bool;
   //    Reset : Bool;
   //    REAC_DELAY { ExternalWritable := 'False'} : Time;
   //    Bypass_ET200 : Bool;
   // END_VAR
   // VAR_OUTPUT
   //    OUT_1 : Bool;
   //    OUT_2 : Bool;
   //    OUT_3 : Bool;
   //    OUT_4 : Bool;
   //    Diag_1 : Bool;
   //    Diag_2 : Bool;
   //    Diag_3 : Bool;
   //    Diag_4 : Bool;
   //    Lamp_1 : Bool;
   //    Lamp_2 : Bool;
   //    Lamp_3 : Bool;
   //    Lamp_4 : Bool;
   // END_VAR
   // VAR
   //    ESTOP_1 { S7_SetPoint := 'True'} : ESTOP1;
   //    ESTOP_2 { S7_SetPoint := 'True'} : ESTOP1;
   //    ESTOP_3 { S7_SetPoint := 'True'} : ESTOP1;
   //    ESTOP_4 { S7_SetPoint := 'True'} : ESTOP1;
   //    TON_1 { ExternalWritable := 'False'} : TON;
   //    TON_2 { ExternalWritable := 'False'} : TON;
   //    TON_3 { ExternalWritable := 'False'} : TON;
   //    TON_4 { ExternalWritable := 'False'} : TON;
   // END_VAR
BEGIN
END_DATA_BLOCK

DATA_BLOCK "n0005-lv008-el001-k30001_SN51_1"   // DB1070, F_DB
VERSION : 0.1
// stored: AutoNumber true, DBAccessibleFromOPCUA true, DBAccessibleFromWebserver true, InstanceOfName 00_Push-Button_Input, InstanceOfType FB
"00_Push-Button_Input"
   // VAR_INPUT
   //    IN_1 : Bool;
   //    IN_2 : Bool;
   //    IN_3 : Bool;
   //    IN_4 : Bool;
   //    ON_Tristate : Bool;
   //    ON_Lamp : Bool;
   //    Reset : Bool;
   //    REAC_DELAY { ExternalWritable := 'False'} : Time;
   //    Bypass_ET200 : Bool;
   // END_VAR
   // VAR_OUTPUT
   //    OUT_1 : Bool;
   //    OUT_2 : Bool;
   //    OUT_3 : Bool;
   //    OUT_4 : Bool;
   //    Diag_1 : Bool;
   //    Diag_2 : Bool;
   //    Diag_3 : Bool;
   //    Diag_4 : Bool;
   //    Lamp_1 : Bool;
   //    Lamp_2 : Bool;
   //    Lamp_3 : Bool;
   //    Lamp_4 : Bool;
   // END_VAR
   // VAR
   //    ESTOP_1 { S7_SetPoint := 'True'} : ESTOP1;
   //    ESTOP_2 { S7_SetPoint := 'True'} : ESTOP1;
   //    ESTOP_3 { S7_SetPoint := 'True'} : ESTOP1;
   //    ESTOP_4 { S7_SetPoint := 'True'} : ESTOP1;
   //    TON_1 { ExternalWritable := 'False'} : TON;
   //    TON_2 { ExternalWritable := 'False'} : TON;
   //    TON_3 { ExternalWritable := 'False'} : TON;
   //    TON_4 { ExternalWritable := 'False'} : TON;
   // END_VAR
BEGIN
END_DATA_BLOCK

DATA_BLOCK "n0006-lv008-el001-k30001_SN51_1"   // DB1071, F_DB
VERSION : 0.1
// stored: AutoNumber true, DBAccessibleFromOPCUA true, DBAccessibleFromWebserver true, InstanceOfName 00_Push-Button_Input, InstanceOfType FB
"00_Push-Button_Input"
   // VAR_INPUT
   //    IN_1 : Bool;
   //    IN_2 : Bool;
   //    IN_3 : Bool;
   //    IN_4 : Bool;
   //    ON_Tristate : Bool;
   //    ON_Lamp : Bool;
   //    Reset : Bool;
   //    REAC_DELAY { ExternalWritable := 'False'} : Time;
   //    Bypass_ET200 : Bool;
   // END_VAR
   // VAR_OUTPUT
   //    OUT_1 : Bool;
   //    OUT_2 : Bool;
   //    OUT_3 : Bool;
   //    OUT_4 : Bool;
   //    Diag_1 : Bool;
   //    Diag_2 : Bool;
   //    Diag_3 : Bool;
   //    Diag_4 : Bool;
   //    Lamp_1 : Bool;
   //    Lamp_2 : Bool;
   //    Lamp_3 : Bool;
   //    Lamp_4 : Bool;
   // END_VAR
   // VAR
   //    ESTOP_1 { S7_SetPoint := 'True'} : ESTOP1;
   //    ESTOP_2 { S7_SetPoint := 'True'} : ESTOP1;
   //    ESTOP_3 { S7_SetPoint := 'True'} : ESTOP1;
   //    ESTOP_4 { S7_SetPoint := 'True'} : ESTOP1;
   //    TON_1 { ExternalWritable := 'False'} : TON;
   //    TON_2 { ExternalWritable := 'False'} : TON;
   //    TON_3 { ExternalWritable := 'False'} : TON;
   //    TON_4 { ExternalWritable := 'False'} : TON;
   // END_VAR
BEGIN
END_DATA_BLOCK

DATA_BLOCK "n0007-icg22-el001-k30001_SN51_1"   // DB1072, F_DB
VERSION : 0.1
// stored: AutoNumber true, DBAccessibleFromOPCUA true, DBAccessibleFromWebserver true, InstanceOfName 00_Push-Button_Input, InstanceOfType FB
"00_Push-Button_Input"
   // VAR_INPUT
   //    IN_1 : Bool;
   //    IN_2 : Bool;
   //    IN_3 : Bool;
   //    IN_4 : Bool;
   //    ON_Tristate : Bool;
   //    ON_Lamp : Bool;
   //    Reset : Bool;
   //    REAC_DELAY { ExternalWritable := 'False'} : Time;
   //    Bypass_ET200 : Bool;
   // END_VAR
   // VAR_OUTPUT
   //    OUT_1 : Bool;
   //    OUT_2 : Bool;
   //    OUT_3 : Bool;
   //    OUT_4 : Bool;
   //    Diag_1 : Bool;
   //    Diag_2 : Bool;
   //    Diag_3 : Bool;
   //    Diag_4 : Bool;
   //    Lamp_1 : Bool;
   //    Lamp_2 : Bool;
   //    Lamp_3 : Bool;
   //    Lamp_4 : Bool;
   // END_VAR
   // VAR
   //    ESTOP_1 { S7_SetPoint := 'True'} : ESTOP1;
   //    ESTOP_2 { S7_SetPoint := 'True'} : ESTOP1;
   //    ESTOP_3 { S7_SetPoint := 'True'} : ESTOP1;
   //    ESTOP_4 { S7_SetPoint := 'True'} : ESTOP1;
   //    TON_1 { ExternalWritable := 'False'} : TON;
   //    TON_2 { ExternalWritable := 'False'} : TON;
   //    TON_3 { ExternalWritable := 'False'} : TON;
   //    TON_4 { ExternalWritable := 'False'} : TON;
   // END_VAR
BEGIN
END_DATA_BLOCK

DATA_BLOCK "n0007-icg22-el001-k30001_SN51_2"   // DB1073, F_DB
VERSION : 0.1
// stored: AutoNumber true, DBAccessibleFromOPCUA true, DBAccessibleFromWebserver true, InstanceOfName 00_Push-Button_Input, InstanceOfType FB
"00_Push-Button_Input"
   // VAR_INPUT
   //    IN_1 : Bool;
   //    IN_2 : Bool;
   //    IN_3 : Bool;
   //    IN_4 : Bool;
   //    ON_Tristate : Bool;
   //    ON_Lamp : Bool;
   //    Reset : Bool;
   //    REAC_DELAY { ExternalWritable := 'False'} : Time;
   //    Bypass_ET200 : Bool;
   // END_VAR
   // VAR_OUTPUT
   //    OUT_1 : Bool;
   //    OUT_2 : Bool;
   //    OUT_3 : Bool;
   //    OUT_4 : Bool;
   //    Diag_1 : Bool;
   //    Diag_2 : Bool;
   //    Diag_3 : Bool;
   //    Diag_4 : Bool;
   //    Lamp_1 : Bool;
   //    Lamp_2 : Bool;
   //    Lamp_3 : Bool;
   //    Lamp_4 : Bool;
   // END_VAR
   // VAR
   //    ESTOP_1 { S7_SetPoint := 'True'} : ESTOP1;
   //    ESTOP_2 { S7_SetPoint := 'True'} : ESTOP1;
   //    ESTOP_3 { S7_SetPoint := 'True'} : ESTOP1;
   //    ESTOP_4 { S7_SetPoint := 'True'} : ESTOP1;
   //    TON_1 { ExternalWritable := 'False'} : TON;
   //    TON_2 { ExternalWritable := 'False'} : TON;
   //    TON_3 { ExternalWritable := 'False'} : TON;
   //    TON_4 { ExternalWritable := 'False'} : TON;
   // END_VAR
BEGIN
END_DATA_BLOCK

DATA_BLOCK "n0008-icg12-el001-k30001_SN51_1"   // DB1074, F_DB
VERSION : 0.1
// stored: AutoNumber true, DBAccessibleFromOPCUA true, DBAccessibleFromWebserver true, InstanceOfName 00_Push-Button_Input, InstanceOfType FB
"00_Push-Button_Input"
   // VAR_INPUT
   //    IN_1 : Bool;
   //    IN_2 : Bool;
   //    IN_3 : Bool;
   //    IN_4 : Bool;
   //    ON_Tristate : Bool;
   //    ON_Lamp : Bool;
   //    Reset : Bool;
   //    REAC_DELAY { ExternalWritable := 'False'} : Time;
   //    Bypass_ET200 : Bool;
   // END_VAR
   // VAR_OUTPUT
   //    OUT_1 : Bool;
   //    OUT_2 : Bool;
   //    OUT_3 : Bool;
   //    OUT_4 : Bool;
   //    Diag_1 : Bool;
   //    Diag_2 : Bool;
   //    Diag_3 : Bool;
   //    Diag_4 : Bool;
   //    Lamp_1 : Bool;
   //    Lamp_2 : Bool;
   //    Lamp_3 : Bool;
   //    Lamp_4 : Bool;
   // END_VAR
   // VAR
   //    ESTOP_1 { S7_SetPoint := 'True'} : ESTOP1;
   //    ESTOP_2 { S7_SetPoint := 'True'} : ESTOP1;
   //    ESTOP_3 { S7_SetPoint := 'True'} : ESTOP1;
   //    ESTOP_4 { S7_SetPoint := 'True'} : ESTOP1;
   //    TON_1 { ExternalWritable := 'False'} : TON;
   //    TON_2 { ExternalWritable := 'False'} : TON;
   //    TON_3 { ExternalWritable := 'False'} : TON;
   //    TON_4 { ExternalWritable := 'False'} : TON;
   // END_VAR
BEGIN
END_DATA_BLOCK

DATA_BLOCK "n0008-icg12-el001-k30001_SN51_2"   // DB1075, F_DB
VERSION : 0.1
// stored: AutoNumber true, DBAccessibleFromOPCUA true, DBAccessibleFromWebserver true, InstanceOfName 00_Push-Button_Input, InstanceOfType FB
"00_Push-Button_Input"
   // VAR_INPUT
   //    IN_1 : Bool;
   //    IN_2 : Bool;
   //    IN_3 : Bool;
   //    IN_4 : Bool;
   //    ON_Tristate : Bool;
   //    ON_Lamp : Bool;
   //    Reset : Bool;
   //    REAC_DELAY { ExternalWritable := 'False'} : Time;
   //    Bypass_ET200 : Bool;
   // END_VAR
   // VAR_OUTPUT
   //    OUT_1 : Bool;
   //    OUT_2 : Bool;
   //    OUT_3 : Bool;
   //    OUT_4 : Bool;
   //    Diag_1 : Bool;
   //    Diag_2 : Bool;
   //    Diag_3 : Bool;
   //    Diag_4 : Bool;
   //    Lamp_1 : Bool;
   //    Lamp_2 : Bool;
   //    Lamp_3 : Bool;
   //    Lamp_4 : Bool;
   // END_VAR
   // VAR
   //    ESTOP_1 { S7_SetPoint := 'True'} : ESTOP1;
   //    ESTOP_2 { S7_SetPoint := 'True'} : ESTOP1;
   //    ESTOP_3 { S7_SetPoint := 'True'} : ESTOP1;
   //    ESTOP_4 { S7_SetPoint := 'True'} : ESTOP1;
   //    TON_1 { ExternalWritable := 'False'} : TON;
   //    TON_2 { ExternalWritable := 'False'} : TON;
   //    TON_3 { ExternalWritable := 'False'} : TON;
   //    TON_4 { ExternalWritable := 'False'} : TON;
   // END_VAR
BEGIN
END_DATA_BLOCK

